// TwinCAT 3 PLC project plc_mrco_vac
// ProgramVersion: 3.1.4022.7
// libraries:
//   LCLS General, * (SLAC)
//   LCLS Vacuum, * (SLAC - LCLS)
//   LCLSVacuumSerialDriverLib, * (SLAC - LCLS)
//   PMPS, * (SLAC - LCLS)
//   Tc2_SerialCom, * (Beckhoff Automation GmbH)
//   Tc2_Standard, * (Beckhoff Automation GmbH)
//   Tc2_System, * (Beckhoff Automation GmbH)
//   Tc3_Module, * (Beckhoff Automation GmbH)
// project tree:
//   / ComTask.TcTTO, PlcTask.TcTTO
//   GVLs/ GVL_COM.TcGVL, GVL_Devices.TcGVL, GVL_PLC_Interfaces.TcGVL, GVL_TC.TcGVL, GVL_Variables.TcGVL
//   POUs/ DIAGNOSTICS.TcPOU, F_Turbo_NC_NO_Valve_Logic.TcPOU, MAIN.TcPOU, PRG_COM.TcPOU, PRG_TC.TcPOU
// real-time tasks:
//   TASK PlcTask: cycle T#10ms, priority 20, ADS port 350
//   TASK ComTask: cycle T#10ms, priority 15, ADS port 351
// I/O:
//   DEVICE Device 1 (EtherCAT), AmsNetId 172.21.132.115.2.1
//     MRCO_PLC_E00_EK1200 [EK1200-5000 EtherCAT Power supply (2A E-Bus)]
//       MRCO_PLC_E01_EL2202
//       MRCO_PLC_E03_EL9184 [EL9184 Potential Connection, 8 x 24V, 8 x Ground]
//       MRCO_PLC_E04_EL6695 [EL6695 EtherCAT Bridge terminal (Primary)]
//       MRCO_PLC_E05_EL9410 [EL9410 E-Bus Power Supplier  (Diagnostics)]
//       MRCO_PLC_E06_EL1004 [EL1004 4Ch. Dig. Input 24V, 3ms]
//       MRCO_PLC_E07_EL2794 [EL2794 4Ch. Dig. Output 24V AC/DC, 2A, short-circuit-proof]
//       MRCO_PLC_E08_EL1004 [EL1004 4Ch. Dig. Input 24V, 3ms]
//       MRCO_PLC_E09_EL2794 [EL2794 4Ch. Dig. Output 24V AC/DC, 2A, short-circuit-proof]
//       MRCO_PLC_E10_EL3318 [EL3318 8Ch. Ana Input Thermocouple (TC)]
//       MRCO_PLC_EXX_EL6070 [EL6070 1Ch. Licensing-Terminal]
//       MRCO_PLC_E11_EL6002 [EL6002 Interface 2Ch. (RS232)]
//       MRCO_PLC_E12_EL6002 [EL6002 Interface 2Ch. (RS232)]
//       MRCO_PLC_E13_EK1122 [EK1122 2 port EtherCAT junction]
//         MRCO_PNL1_EP01_EP2338-0002 [EP2338-0002 8 Ch. Dig. Input/Output 24V, 0,5A, M12]
//         MRCO_PNL1_EP02_EP2624-0002 [EP2624-0002 4Ch. Relay Output, NO (125V AC / 30V DC)]
//         MRCO_PNL1_EP03_EP6002-0002 [EP6002-0002 Interface (RS232/422/485)]
//         MRCO_PNL1_EP04_EP3174-0002 [EP3174-0002 4Ch. Ana. Input +/-10V, 0-10V, 0/4-20mA configurable]
//         MRCO_PNL1_EP05_EP3174-0002 [EP3174-0002 4Ch. Ana. Input +/-10V, 0-10V, 0/4-20mA configurable]
//         MRCO_PNL1_EP06_EP2624-0002
//         MRCO_PNL1_EP07_EP2338-0002 [EP2338-0002 8 Ch. Dig. Input/Output 24V, 0,5A, M12]
//         MRCO_PNL1_EP08_EP2338-0002
//         MRCO_DRL_03 (EK1100) [EK1100 EtherCAT Coupler (2A E-Bus)]
//           MRCO_DRL_03_E01_EL1004
//           MRCO_DRL_03_E02_EL2004 [EL2004 4Ch. Dig. Output 24V, 0.5A]
//           MRCO_DRL_03_E03_EL1004
//           MRCO_DRL_03_E04_EL1004 [EL1004 4Ch. Dig. Input 24V, 3ms]
//           MRCO_DRL_03_E05_EL6001 [EL6001 Interface (RS232)]
//           MRCO_DRL_03_E06_EL2794
//           MRCO_DRL_03_E07_EL1084 [EL1084 4Ch. Dig. Input 24V, 3ms, negative]
//           MRCO_DRL_03_E08_EL9184 [EL9184 Potential Connection, 8 x 24V, 8 x Ground]
//           MRCO_DRL_03_E09_EL9070 [EL9070 Shield terminal]
//           MRCO_DRL_03_E10_EL3174-0002 [EL3174-0002 4Ch. Ana. Input +/-10V, +/-20mA 16 Bit, Isolated Channels]
//           Term 54 (EL9011) [EL9011 End Terminal]
//         VCN_1_VAT590 [590 - All-metal variable leak valve]
// variable links:
//   plc_mrco_vac Instance <-> Device 1 (EtherCAT)/MRCO_PLC_E00_EK1200/MRCO_PLC_E04_EL6695
//     PlcTask Inputs/GVL_PLC_Interfaces.sHUTCH_PLC_NAME <-> IO Inputs/HUTCH_PLC_NAME
//     PlcTask Inputs/GVL_PLC_Interfaces.xEcatBridge_External_device_not_connected <-> SYNC Inputs/External device not connected
//     PlcTask Inputs/GVL_PLC_Interfaces.xEcatBridge_TxPDO_state <-> SYNC Inputs/TxPDO state
//     PlcTask Inputs/GVL_PLC_Interfaces.xEcatBridge_WcState <-> WcState/WcState
//     PlcTask Inputs/GVL_PLC_Interfaces.xTMO_ROUGH1_VRC_01_OPEN_LS <-> IO Inputs/TMO_ROUGH1_VRC_01_OPEN_LS
//     PlcTask Inputs/GVL_PLC_Interfaces.xTMO_ROUGH2_VRC_01_OPEN_LS <-> IO Inputs/TMO_ROUGH2_VRC_01_OPEN_LS
//     PlcTask Outputs/GVL_PLC_Interfaces.rIP1_MAIN_rPRESS <-> IO Outputs/IP1_MAIN_rPRESS
//     PlcTask Outputs/GVL_PLC_Interfaces.sENDSTATION_PLC_NAME <-> IO Outputs/ENDSTATION_PLC_NAME
//     PlcTask Outputs/GVL_PLC_Interfaces.xIP1_HV_SAFETY_ENABLE <-> IO Outputs/IP1_HV_SAFETY_ENABLE
//     PlcTask Outputs/GVL_PLC_Interfaces.xIP1_MAIN_xAT_VAC <-> IO Outputs/IP1_MAIN_xAT_VAC
//     PlcTask Outputs/GVL_PLC_Interfaces.xIP1_MAIN_xPRESS_OK <-> IO Outputs/IP1_MAIN_xPRESS_OK
//     PlcTask Outputs/GVL_PLC_Interfaces.xIP1_ROUGH_VRC_01_OPEN_LS <-> IO Outputs/IP1_ROUGH_VRC_01_OPEN_LS
//     PlcTask Outputs/GVL_PLC_Interfaces.xIP1_ROUGH_VRC_02_OPEN_LS <-> IO Outputs/IP1_ROUGH_VRC_02_OPEN_LS
//     PlcTask Outputs/GVL_PLC_Interfaces.xIP1_ROUGH_VRC_03_OPEN_LS <-> IO Outputs/IP1_ROUGH_VRC_03_OPEN_LS
//     PlcTask Outputs/GVL_PLC_Interfaces.xIP1_TURBOS_ALL_AtSpd <-> IO Outputs/IP1_TURBOS_ALL_AtSpd
//   plc_mrco_vac Instance <-> Device 1 (EtherCAT)/MRCO_PLC_E00_EK1200/MRCO_PLC_E06_EL1004
//     PlcTask Inputs/GVL_Devices.MRCO_MAIN_PTM_01.i_xAtSpd <-> Channel 2/Input
//     PlcTask Inputs/GVL_Devices.MRCO_MAIN_PTM_02.i_xAtSpd <-> Channel 4/Input
//     PlcTask Inputs/GVL_Devices.MRCO_MAIN_PTM_01.i_xFaultNC <-> Channel 1/Input
//     PlcTask Inputs/GVL_Devices.MRCO_MAIN_PTM_02.i_xFaultNC <-> Channel 3/Input
//   plc_mrco_vac Instance <-> Device 1 (EtherCAT)/MRCO_PLC_E00_EK1200/MRCO_PLC_E07_EL2794
//     PlcTask Outputs/GVL_Devices.MRCO_MAIN_PTM_01.q_RunDO <-> Channel 1/Output
//     PlcTask Outputs/GVL_Devices.MRCO_MAIN_PTM_02.q_RunDO <-> Channel 3/Output
//     PlcTask Outputs/GVL_Devices.MRCO_MAIN_PTM_03.q_RunDO <-> Channel 2/Output
//     PlcTask Outputs/GVL_Devices.MRCO_MAIN_PTM_04.q_RunDO <-> Channel 4/Output
//   plc_mrco_vac Instance <-> Device 1 (EtherCAT)/MRCO_PLC_E00_EK1200/MRCO_PLC_E08_EL1004
//     PlcTask Inputs/GVL_Devices.MRCO_MAIN_PTM_03.i_xAtSpd <-> Channel 2/Input
//     PlcTask Inputs/GVL_Devices.MRCO_MAIN_PTM_04.i_xAtSpd <-> Channel 4/Input
//     PlcTask Inputs/GVL_Devices.MRCO_MAIN_PTM_03.i_xFaultNC <-> Channel 1/Input
//     PlcTask Inputs/GVL_Devices.MRCO_MAIN_PTM_04.i_xFaultNC <-> Channel 3/Input
//   plc_mrco_vac Instance <-> Device 1 (EtherCAT)/MRCO_PLC_E00_EK1200/MRCO_PLC_E09_EL2794
//     PlcTask Outputs/GVL_PLC_Interfaces.xHighVoltageSafteyLoopEnable <-> Channel 1/Output
//   plc_mrco_vac Instance <-> Device 1 (EtherCAT)/MRCO_PLC_E00_EK1200/MRCO_PLC_E10_EL3318
//     PlcTask Inputs/GVL_TC.TC_01.bError <-> TC Channel 1/Status/Error
//     PlcTask Inputs/GVL_TC.TC_02.bError <-> TC Channel 2/Status/Error
//     PlcTask Inputs/GVL_TC.TC_03.bError <-> TC Channel 3/Status/Error
//     PlcTask Inputs/GVL_TC.TC_04.bError <-> TC Channel 4/Status/Error
//     PlcTask Inputs/GVL_TC.TC_05.bError <-> TC Channel 5/Status/Error
//     PlcTask Inputs/GVL_TC.TC_06.bError <-> TC Channel 6/Status/Error
//     PlcTask Inputs/GVL_TC.TC_07.bError <-> TC Channel 7/Status/Error
//     PlcTask Inputs/GVL_TC.TC_08.bError <-> TC Channel 8/Status/Error
//     PlcTask Inputs/GVL_TC.TC_01.bOverrange <-> TC Channel 1/Status/Overrange
//     PlcTask Inputs/GVL_TC.TC_02.bOverrange <-> TC Channel 2/Status/Overrange
//     PlcTask Inputs/GVL_TC.TC_03.bOverrange <-> TC Channel 3/Status/Overrange
//     PlcTask Inputs/GVL_TC.TC_04.bOverrange <-> TC Channel 4/Status/Overrange
//     PlcTask Inputs/GVL_TC.TC_05.bOverrange <-> TC Channel 5/Status/Overrange
//     PlcTask Inputs/GVL_TC.TC_06.bOverrange <-> TC Channel 6/Status/Overrange
//     PlcTask Inputs/GVL_TC.TC_07.bOverrange <-> TC Channel 7/Status/Overrange
//     PlcTask Inputs/GVL_TC.TC_08.bOverrange <-> TC Channel 8/Status/Overrange
//     PlcTask Inputs/GVL_TC.TC_01.bUnderrange <-> TC Channel 1/Status/Underrange
//     PlcTask Inputs/GVL_TC.TC_02.bUnderrange <-> TC Channel 2/Status/Underrange
//     PlcTask Inputs/GVL_TC.TC_03.bUnderrange <-> TC Channel 3/Status/Underrange
//     PlcTask Inputs/GVL_TC.TC_04.bUnderrange <-> TC Channel 4/Status/Underrange
//     PlcTask Inputs/GVL_TC.TC_05.bUnderrange <-> TC Channel 5/Status/Underrange
//     PlcTask Inputs/GVL_TC.TC_06.bUnderrange <-> TC Channel 6/Status/Underrange
//     PlcTask Inputs/GVL_TC.TC_07.bUnderrange <-> TC Channel 7/Status/Underrange
//     PlcTask Inputs/GVL_TC.TC_08.bUnderrange <-> TC Channel 8/Status/Underrange
//     PlcTask Inputs/GVL_TC.TC_01.iRaw <-> TC Channel 1/Value
//     PlcTask Inputs/GVL_TC.TC_02.iRaw <-> TC Channel 2/Value
//     PlcTask Inputs/GVL_TC.TC_03.iRaw <-> TC Channel 3/Value
//     PlcTask Inputs/GVL_TC.TC_04.iRaw <-> TC Channel 4/Value
//     PlcTask Inputs/GVL_TC.TC_05.iRaw <-> TC Channel 5/Value
//     PlcTask Inputs/GVL_TC.TC_06.iRaw <-> TC Channel 6/Value
//     PlcTask Inputs/GVL_TC.TC_07.iRaw <-> TC Channel 7/Value
//     PlcTask Inputs/GVL_TC.TC_08.iRaw <-> TC Channel 8/Value
//   plc_mrco_vac Instance <-> Device 1 (EtherCAT)/MRCO_PLC_E00_EK1200/MRCO_PLC_E11_EL6002
//     ComTask Inputs/GVL_COM.stComIn_MRCO_MAIN_PTM_01/D[0] <-> COM TxPDO-Map Inputs Channel 1/Data In 0
//     ComTask Inputs/GVL_COM.stComIn_MRCO_MAIN_PTM_01/D[10] <-> COM TxPDO-Map Inputs Channel 1/Data In 10
//     ComTask Inputs/GVL_COM.stComIn_MRCO_MAIN_PTM_01/D[11] <-> COM TxPDO-Map Inputs Channel 1/Data In 11
//     ComTask Inputs/GVL_COM.stComIn_MRCO_MAIN_PTM_01/D[12] <-> COM TxPDO-Map Inputs Channel 1/Data In 12
//     ComTask Inputs/GVL_COM.stComIn_MRCO_MAIN_PTM_01/D[13] <-> COM TxPDO-Map Inputs Channel 1/Data In 13
//     ComTask Inputs/GVL_COM.stComIn_MRCO_MAIN_PTM_01/D[14] <-> COM TxPDO-Map Inputs Channel 1/Data In 14
//     ComTask Inputs/GVL_COM.stComIn_MRCO_MAIN_PTM_01/D[15] <-> COM TxPDO-Map Inputs Channel 1/Data In 15
//     ComTask Inputs/GVL_COM.stComIn_MRCO_MAIN_PTM_01/D[16] <-> COM TxPDO-Map Inputs Channel 1/Data In 16
//     ComTask Inputs/GVL_COM.stComIn_MRCO_MAIN_PTM_01/D[17] <-> COM TxPDO-Map Inputs Channel 1/Data In 17
//     ComTask Inputs/GVL_COM.stComIn_MRCO_MAIN_PTM_01/D[18] <-> COM TxPDO-Map Inputs Channel 1/Data In 18
//     ComTask Inputs/GVL_COM.stComIn_MRCO_MAIN_PTM_01/D[19] <-> COM TxPDO-Map Inputs Channel 1/Data In 19
//     ComTask Inputs/GVL_COM.stComIn_MRCO_MAIN_PTM_01/D[1] <-> COM TxPDO-Map Inputs Channel 1/Data In 1
//     ComTask Inputs/GVL_COM.stComIn_MRCO_MAIN_PTM_01/D[20] <-> COM TxPDO-Map Inputs Channel 1/Data In 20
//     ComTask Inputs/GVL_COM.stComIn_MRCO_MAIN_PTM_01/D[21] <-> COM TxPDO-Map Inputs Channel 1/Data In 21
//     ComTask Inputs/GVL_COM.stComIn_MRCO_MAIN_PTM_01/D[2] <-> COM TxPDO-Map Inputs Channel 1/Data In 2
//     ComTask Inputs/GVL_COM.stComIn_MRCO_MAIN_PTM_01/D[3] <-> COM TxPDO-Map Inputs Channel 1/Data In 3
//     ComTask Inputs/GVL_COM.stComIn_MRCO_MAIN_PTM_01/D[4] <-> COM TxPDO-Map Inputs Channel 1/Data In 4
//     ComTask Inputs/GVL_COM.stComIn_MRCO_MAIN_PTM_01/D[5] <-> COM TxPDO-Map Inputs Channel 1/Data In 5
//     ComTask Inputs/GVL_COM.stComIn_MRCO_MAIN_PTM_01/D[6] <-> COM TxPDO-Map Inputs Channel 1/Data In 6
//     ComTask Inputs/GVL_COM.stComIn_MRCO_MAIN_PTM_01/D[7] <-> COM TxPDO-Map Inputs Channel 1/Data In 7
//     ComTask Inputs/GVL_COM.stComIn_MRCO_MAIN_PTM_01/D[8] <-> COM TxPDO-Map Inputs Channel 1/Data In 8
//     ComTask Inputs/GVL_COM.stComIn_MRCO_MAIN_PTM_01/D[9] <-> COM TxPDO-Map Inputs Channel 1/Data In 9
//     ComTask Inputs/GVL_COM.stComIn_MRCO_MAIN_PTM_03/D[0] <-> COM TxPDO-Map Inputs Channel 2/Data In 0
//     ComTask Inputs/GVL_COM.stComIn_MRCO_MAIN_PTM_03/D[10] <-> COM TxPDO-Map Inputs Channel 2/Data In 10
//     ComTask Inputs/GVL_COM.stComIn_MRCO_MAIN_PTM_03/D[11] <-> COM TxPDO-Map Inputs Channel 2/Data In 11
//     ComTask Inputs/GVL_COM.stComIn_MRCO_MAIN_PTM_03/D[12] <-> COM TxPDO-Map Inputs Channel 2/Data In 12
//     ComTask Inputs/GVL_COM.stComIn_MRCO_MAIN_PTM_03/D[13] <-> COM TxPDO-Map Inputs Channel 2/Data In 13
//     ComTask Inputs/GVL_COM.stComIn_MRCO_MAIN_PTM_03/D[14] <-> COM TxPDO-Map Inputs Channel 2/Data In 14
//     ComTask Inputs/GVL_COM.stComIn_MRCO_MAIN_PTM_03/D[15] <-> COM TxPDO-Map Inputs Channel 2/Data In 15
//     ComTask Inputs/GVL_COM.stComIn_MRCO_MAIN_PTM_03/D[16] <-> COM TxPDO-Map Inputs Channel 2/Data In 16
//     ComTask Inputs/GVL_COM.stComIn_MRCO_MAIN_PTM_03/D[17] <-> COM TxPDO-Map Inputs Channel 2/Data In 17
//     ComTask Inputs/GVL_COM.stComIn_MRCO_MAIN_PTM_03/D[18] <-> COM TxPDO-Map Inputs Channel 2/Data In 18
//     ComTask Inputs/GVL_COM.stComIn_MRCO_MAIN_PTM_03/D[19] <-> COM TxPDO-Map Inputs Channel 2/Data In 19
//     ComTask Inputs/GVL_COM.stComIn_MRCO_MAIN_PTM_03/D[1] <-> COM TxPDO-Map Inputs Channel 2/Data In 1
//     ComTask Inputs/GVL_COM.stComIn_MRCO_MAIN_PTM_03/D[20] <-> COM TxPDO-Map Inputs Channel 2/Data In 20
//     ComTask Inputs/GVL_COM.stComIn_MRCO_MAIN_PTM_03/D[21] <-> COM TxPDO-Map Inputs Channel 2/Data In 21
//     ComTask Inputs/GVL_COM.stComIn_MRCO_MAIN_PTM_03/D[2] <-> COM TxPDO-Map Inputs Channel 2/Data In 2
//     ComTask Inputs/GVL_COM.stComIn_MRCO_MAIN_PTM_03/D[3] <-> COM TxPDO-Map Inputs Channel 2/Data In 3
//     ComTask Inputs/GVL_COM.stComIn_MRCO_MAIN_PTM_03/D[4] <-> COM TxPDO-Map Inputs Channel 2/Data In 4
//     ComTask Inputs/GVL_COM.stComIn_MRCO_MAIN_PTM_03/D[5] <-> COM TxPDO-Map Inputs Channel 2/Data In 5
//     ComTask Inputs/GVL_COM.stComIn_MRCO_MAIN_PTM_03/D[6] <-> COM TxPDO-Map Inputs Channel 2/Data In 6
//     ComTask Inputs/GVL_COM.stComIn_MRCO_MAIN_PTM_03/D[7] <-> COM TxPDO-Map Inputs Channel 2/Data In 7
//     ComTask Inputs/GVL_COM.stComIn_MRCO_MAIN_PTM_03/D[8] <-> COM TxPDO-Map Inputs Channel 2/Data In 8
//     ComTask Inputs/GVL_COM.stComIn_MRCO_MAIN_PTM_03/D[9] <-> COM TxPDO-Map Inputs Channel 2/Data In 9
//     ComTask Inputs/GVL_COM.stComIn_MRCO_MAIN_PTM_01/Status <-> COM TxPDO-Map Inputs Channel 1/Status
//     ComTask Inputs/GVL_COM.stComIn_MRCO_MAIN_PTM_03/Status <-> COM TxPDO-Map Inputs Channel 2/Status
//     ComTask Outputs/GVL_COM.stComOut_MRCO_MAIN_PTM_01/Ctrl <-> COM RxPDO-Map Outputs Channel 1/Ctrl
//     ComTask Outputs/GVL_COM.stComOut_MRCO_MAIN_PTM_03/Ctrl <-> COM RxPDO-Map Outputs Channel 2/Ctrl
//     ComTask Outputs/GVL_COM.stComOut_MRCO_MAIN_PTM_01/D[0] <-> COM RxPDO-Map Outputs Channel 1/Data Out 0
//     ComTask Outputs/GVL_COM.stComOut_MRCO_MAIN_PTM_01/D[10] <-> COM RxPDO-Map Outputs Channel 1/Data Out 10
//     ComTask Outputs/GVL_COM.stComOut_MRCO_MAIN_PTM_01/D[11] <-> COM RxPDO-Map Outputs Channel 1/Data Out 11
//     ComTask Outputs/GVL_COM.stComOut_MRCO_MAIN_PTM_01/D[12] <-> COM RxPDO-Map Outputs Channel 1/Data Out 12
//     ComTask Outputs/GVL_COM.stComOut_MRCO_MAIN_PTM_01/D[13] <-> COM RxPDO-Map Outputs Channel 1/Data Out 13
//     ComTask Outputs/GVL_COM.stComOut_MRCO_MAIN_PTM_01/D[14] <-> COM RxPDO-Map Outputs Channel 1/Data Out 14
//     ComTask Outputs/GVL_COM.stComOut_MRCO_MAIN_PTM_01/D[15] <-> COM RxPDO-Map Outputs Channel 1/Data Out 15
//     ComTask Outputs/GVL_COM.stComOut_MRCO_MAIN_PTM_01/D[16] <-> COM RxPDO-Map Outputs Channel 1/Data Out 16
//     ComTask Outputs/GVL_COM.stComOut_MRCO_MAIN_PTM_01/D[17] <-> COM RxPDO-Map Outputs Channel 1/Data Out 17
//     ComTask Outputs/GVL_COM.stComOut_MRCO_MAIN_PTM_01/D[18] <-> COM RxPDO-Map Outputs Channel 1/Data Out 18
//     ComTask Outputs/GVL_COM.stComOut_MRCO_MAIN_PTM_01/D[19] <-> COM RxPDO-Map Outputs Channel 1/Data Out 19
//     ComTask Outputs/GVL_COM.stComOut_MRCO_MAIN_PTM_01/D[1] <-> COM RxPDO-Map Outputs Channel 1/Data Out 1
//     ComTask Outputs/GVL_COM.stComOut_MRCO_MAIN_PTM_01/D[20] <-> COM RxPDO-Map Outputs Channel 1/Data Out 20
//     ComTask Outputs/GVL_COM.stComOut_MRCO_MAIN_PTM_01/D[21] <-> COM RxPDO-Map Outputs Channel 1/Data Out 21
//     ComTask Outputs/GVL_COM.stComOut_MRCO_MAIN_PTM_01/D[2] <-> COM RxPDO-Map Outputs Channel 1/Data Out 2
//     ComTask Outputs/GVL_COM.stComOut_MRCO_MAIN_PTM_01/D[3] <-> COM RxPDO-Map Outputs Channel 1/Data Out 3
//     ComTask Outputs/GVL_COM.stComOut_MRCO_MAIN_PTM_01/D[4] <-> COM RxPDO-Map Outputs Channel 1/Data Out 4
//     ComTask Outputs/GVL_COM.stComOut_MRCO_MAIN_PTM_01/D[5] <-> COM RxPDO-Map Outputs Channel 1/Data Out 5
//     ComTask Outputs/GVL_COM.stComOut_MRCO_MAIN_PTM_01/D[6] <-> COM RxPDO-Map Outputs Channel 1/Data Out 6
//     ComTask Outputs/GVL_COM.stComOut_MRCO_MAIN_PTM_01/D[7] <-> COM RxPDO-Map Outputs Channel 1/Data Out 7
//     ComTask Outputs/GVL_COM.stComOut_MRCO_MAIN_PTM_01/D[8] <-> COM RxPDO-Map Outputs Channel 1/Data Out 8
//     ComTask Outputs/GVL_COM.stComOut_MRCO_MAIN_PTM_01/D[9] <-> COM RxPDO-Map Outputs Channel 1/Data Out 9
//     ComTask Outputs/GVL_COM.stComOut_MRCO_MAIN_PTM_03/D[0] <-> COM RxPDO-Map Outputs Channel 2/Data Out 0
//     ComTask Outputs/GVL_COM.stComOut_MRCO_MAIN_PTM_03/D[10] <-> COM RxPDO-Map Outputs Channel 2/Data Out 10
//     ComTask Outputs/GVL_COM.stComOut_MRCO_MAIN_PTM_03/D[11] <-> COM RxPDO-Map Outputs Channel 2/Data Out 11
//     ComTask Outputs/GVL_COM.stComOut_MRCO_MAIN_PTM_03/D[12] <-> COM RxPDO-Map Outputs Channel 2/Data Out 12
//     ComTask Outputs/GVL_COM.stComOut_MRCO_MAIN_PTM_03/D[13] <-> COM RxPDO-Map Outputs Channel 2/Data Out 13
//     ComTask Outputs/GVL_COM.stComOut_MRCO_MAIN_PTM_03/D[14] <-> COM RxPDO-Map Outputs Channel 2/Data Out 14
//     ComTask Outputs/GVL_COM.stComOut_MRCO_MAIN_PTM_03/D[15] <-> COM RxPDO-Map Outputs Channel 2/Data Out 15
//     ComTask Outputs/GVL_COM.stComOut_MRCO_MAIN_PTM_03/D[16] <-> COM RxPDO-Map Outputs Channel 2/Data Out 16
//     ComTask Outputs/GVL_COM.stComOut_MRCO_MAIN_PTM_03/D[17] <-> COM RxPDO-Map Outputs Channel 2/Data Out 17
//     ComTask Outputs/GVL_COM.stComOut_MRCO_MAIN_PTM_03/D[18] <-> COM RxPDO-Map Outputs Channel 2/Data Out 18
//     ComTask Outputs/GVL_COM.stComOut_MRCO_MAIN_PTM_03/D[19] <-> COM RxPDO-Map Outputs Channel 2/Data Out 19
//     ComTask Outputs/GVL_COM.stComOut_MRCO_MAIN_PTM_03/D[1] <-> COM RxPDO-Map Outputs Channel 2/Data Out 1
//     ComTask Outputs/GVL_COM.stComOut_MRCO_MAIN_PTM_03/D[20] <-> COM RxPDO-Map Outputs Channel 2/Data Out 20
//     ComTask Outputs/GVL_COM.stComOut_MRCO_MAIN_PTM_03/D[21] <-> COM RxPDO-Map Outputs Channel 2/Data Out 21
//     ComTask Outputs/GVL_COM.stComOut_MRCO_MAIN_PTM_03/D[2] <-> COM RxPDO-Map Outputs Channel 2/Data Out 2
//     ComTask Outputs/GVL_COM.stComOut_MRCO_MAIN_PTM_03/D[3] <-> COM RxPDO-Map Outputs Channel 2/Data Out 3
//     ComTask Outputs/GVL_COM.stComOut_MRCO_MAIN_PTM_03/D[4] <-> COM RxPDO-Map Outputs Channel 2/Data Out 4
//     ComTask Outputs/GVL_COM.stComOut_MRCO_MAIN_PTM_03/D[5] <-> COM RxPDO-Map Outputs Channel 2/Data Out 5
//     ComTask Outputs/GVL_COM.stComOut_MRCO_MAIN_PTM_03/D[6] <-> COM RxPDO-Map Outputs Channel 2/Data Out 6
//     ComTask Outputs/GVL_COM.stComOut_MRCO_MAIN_PTM_03/D[7] <-> COM RxPDO-Map Outputs Channel 2/Data Out 7
//     ComTask Outputs/GVL_COM.stComOut_MRCO_MAIN_PTM_03/D[8] <-> COM RxPDO-Map Outputs Channel 2/Data Out 8
//     ComTask Outputs/GVL_COM.stComOut_MRCO_MAIN_PTM_03/D[9] <-> COM RxPDO-Map Outputs Channel 2/Data Out 9
//   plc_mrco_vac Instance <-> Device 1 (EtherCAT)/MRCO_PLC_E00_EK1200/MRCO_PLC_E12_EL6002
//     ComTask Inputs/GVL_COM.stComIn_MRCO_MAIN_PTM_02/D[0] <-> COM TxPDO-Map Inputs Channel 1/Data In 0
//     ComTask Inputs/GVL_COM.stComIn_MRCO_MAIN_PTM_02/D[10] <-> COM TxPDO-Map Inputs Channel 1/Data In 10
//     ComTask Inputs/GVL_COM.stComIn_MRCO_MAIN_PTM_02/D[11] <-> COM TxPDO-Map Inputs Channel 1/Data In 11
//     ComTask Inputs/GVL_COM.stComIn_MRCO_MAIN_PTM_02/D[12] <-> COM TxPDO-Map Inputs Channel 1/Data In 12
//     ComTask Inputs/GVL_COM.stComIn_MRCO_MAIN_PTM_02/D[13] <-> COM TxPDO-Map Inputs Channel 1/Data In 13
//     ComTask Inputs/GVL_COM.stComIn_MRCO_MAIN_PTM_02/D[14] <-> COM TxPDO-Map Inputs Channel 1/Data In 14
//     ComTask Inputs/GVL_COM.stComIn_MRCO_MAIN_PTM_02/D[15] <-> COM TxPDO-Map Inputs Channel 1/Data In 15
//     ComTask Inputs/GVL_COM.stComIn_MRCO_MAIN_PTM_02/D[16] <-> COM TxPDO-Map Inputs Channel 1/Data In 16
//     ComTask Inputs/GVL_COM.stComIn_MRCO_MAIN_PTM_02/D[17] <-> COM TxPDO-Map Inputs Channel 1/Data In 17
//     ComTask Inputs/GVL_COM.stComIn_MRCO_MAIN_PTM_02/D[18] <-> COM TxPDO-Map Inputs Channel 1/Data In 18
//     ComTask Inputs/GVL_COM.stComIn_MRCO_MAIN_PTM_02/D[19] <-> COM TxPDO-Map Inputs Channel 1/Data In 19
//     ComTask Inputs/GVL_COM.stComIn_MRCO_MAIN_PTM_02/D[1] <-> COM TxPDO-Map Inputs Channel 1/Data In 1
//     ComTask Inputs/GVL_COM.stComIn_MRCO_MAIN_PTM_02/D[20] <-> COM TxPDO-Map Inputs Channel 1/Data In 20
//     ComTask Inputs/GVL_COM.stComIn_MRCO_MAIN_PTM_02/D[21] <-> COM TxPDO-Map Inputs Channel 1/Data In 21
//     ComTask Inputs/GVL_COM.stComIn_MRCO_MAIN_PTM_02/D[2] <-> COM TxPDO-Map Inputs Channel 1/Data In 2
//     ComTask Inputs/GVL_COM.stComIn_MRCO_MAIN_PTM_02/D[3] <-> COM TxPDO-Map Inputs Channel 1/Data In 3
//     ComTask Inputs/GVL_COM.stComIn_MRCO_MAIN_PTM_02/D[4] <-> COM TxPDO-Map Inputs Channel 1/Data In 4
//     ComTask Inputs/GVL_COM.stComIn_MRCO_MAIN_PTM_02/D[5] <-> COM TxPDO-Map Inputs Channel 1/Data In 5
//     ComTask Inputs/GVL_COM.stComIn_MRCO_MAIN_PTM_02/D[6] <-> COM TxPDO-Map Inputs Channel 1/Data In 6
//     ComTask Inputs/GVL_COM.stComIn_MRCO_MAIN_PTM_02/D[7] <-> COM TxPDO-Map Inputs Channel 1/Data In 7
//     ComTask Inputs/GVL_COM.stComIn_MRCO_MAIN_PTM_02/D[8] <-> COM TxPDO-Map Inputs Channel 1/Data In 8
//     ComTask Inputs/GVL_COM.stComIn_MRCO_MAIN_PTM_02/D[9] <-> COM TxPDO-Map Inputs Channel 1/Data In 9
//     ComTask Inputs/GVL_COM.stComIn_MRCO_MAIN_PTM_04/D[0] <-> COM TxPDO-Map Inputs Channel 2/Data In 0
//     ComTask Inputs/GVL_COM.stComIn_MRCO_MAIN_PTM_04/D[10] <-> COM TxPDO-Map Inputs Channel 2/Data In 10
//     ComTask Inputs/GVL_COM.stComIn_MRCO_MAIN_PTM_04/D[11] <-> COM TxPDO-Map Inputs Channel 2/Data In 11
//     ComTask Inputs/GVL_COM.stComIn_MRCO_MAIN_PTM_04/D[12] <-> COM TxPDO-Map Inputs Channel 2/Data In 12
//     ComTask Inputs/GVL_COM.stComIn_MRCO_MAIN_PTM_04/D[13] <-> COM TxPDO-Map Inputs Channel 2/Data In 13
//     ComTask Inputs/GVL_COM.stComIn_MRCO_MAIN_PTM_04/D[14] <-> COM TxPDO-Map Inputs Channel 2/Data In 14
//     ComTask Inputs/GVL_COM.stComIn_MRCO_MAIN_PTM_04/D[15] <-> COM TxPDO-Map Inputs Channel 2/Data In 15
//     ComTask Inputs/GVL_COM.stComIn_MRCO_MAIN_PTM_04/D[16] <-> COM TxPDO-Map Inputs Channel 2/Data In 16
//     ComTask Inputs/GVL_COM.stComIn_MRCO_MAIN_PTM_04/D[17] <-> COM TxPDO-Map Inputs Channel 2/Data In 17
//     ComTask Inputs/GVL_COM.stComIn_MRCO_MAIN_PTM_04/D[18] <-> COM TxPDO-Map Inputs Channel 2/Data In 18
//     ComTask Inputs/GVL_COM.stComIn_MRCO_MAIN_PTM_04/D[19] <-> COM TxPDO-Map Inputs Channel 2/Data In 19
//     ComTask Inputs/GVL_COM.stComIn_MRCO_MAIN_PTM_04/D[1] <-> COM TxPDO-Map Inputs Channel 2/Data In 1
//     ComTask Inputs/GVL_COM.stComIn_MRCO_MAIN_PTM_04/D[20] <-> COM TxPDO-Map Inputs Channel 2/Data In 20
//     ComTask Inputs/GVL_COM.stComIn_MRCO_MAIN_PTM_04/D[21] <-> COM TxPDO-Map Inputs Channel 2/Data In 21
//     ComTask Inputs/GVL_COM.stComIn_MRCO_MAIN_PTM_04/D[2] <-> COM TxPDO-Map Inputs Channel 2/Data In 2
//     ComTask Inputs/GVL_COM.stComIn_MRCO_MAIN_PTM_04/D[3] <-> COM TxPDO-Map Inputs Channel 2/Data In 3
//     ComTask Inputs/GVL_COM.stComIn_MRCO_MAIN_PTM_04/D[4] <-> COM TxPDO-Map Inputs Channel 2/Data In 4
//     ComTask Inputs/GVL_COM.stComIn_MRCO_MAIN_PTM_04/D[5] <-> COM TxPDO-Map Inputs Channel 2/Data In 5
//     ComTask Inputs/GVL_COM.stComIn_MRCO_MAIN_PTM_04/D[6] <-> COM TxPDO-Map Inputs Channel 2/Data In 6
//     ComTask Inputs/GVL_COM.stComIn_MRCO_MAIN_PTM_04/D[7] <-> COM TxPDO-Map Inputs Channel 2/Data In 7
//     ComTask Inputs/GVL_COM.stComIn_MRCO_MAIN_PTM_04/D[8] <-> COM TxPDO-Map Inputs Channel 2/Data In 8
//     ComTask Inputs/GVL_COM.stComIn_MRCO_MAIN_PTM_04/D[9] <-> COM TxPDO-Map Inputs Channel 2/Data In 9
//     ComTask Inputs/GVL_COM.stComIn_MRCO_MAIN_PTM_02/Status <-> COM TxPDO-Map Inputs Channel 1/Status
//     ComTask Inputs/GVL_COM.stComIn_MRCO_MAIN_PTM_04/Status <-> COM TxPDO-Map Inputs Channel 2/Status
//     ComTask Outputs/GVL_COM.stComOut_MRCO_MAIN_PTM_02/Ctrl <-> COM RxPDO-Map Outputs Channel 1/Ctrl
//     ComTask Outputs/GVL_COM.stComOut_MRCO_MAIN_PTM_04/Ctrl <-> COM RxPDO-Map Outputs Channel 2/Ctrl
//     ComTask Outputs/GVL_COM.stComOut_MRCO_MAIN_PTM_02/D[10] <-> COM RxPDO-Map Outputs Channel 1/Data Out 10
//     ComTask Outputs/GVL_COM.stComOut_MRCO_MAIN_PTM_02/D[11] <-> COM RxPDO-Map Outputs Channel 1/Data Out 11
//     ComTask Outputs/GVL_COM.stComOut_MRCO_MAIN_PTM_02/D[12] <-> COM RxPDO-Map Outputs Channel 1/Data Out 12
//     ComTask Outputs/GVL_COM.stComOut_MRCO_MAIN_PTM_02/D[13] <-> COM RxPDO-Map Outputs Channel 1/Data Out 13
//     ComTask Outputs/GVL_COM.stComOut_MRCO_MAIN_PTM_02/D[14] <-> COM RxPDO-Map Outputs Channel 1/Data Out 14
//     ComTask Outputs/GVL_COM.stComOut_MRCO_MAIN_PTM_02/D[15] <-> COM RxPDO-Map Outputs Channel 1/Data Out 15
//     ComTask Outputs/GVL_COM.stComOut_MRCO_MAIN_PTM_02/D[16] <-> COM RxPDO-Map Outputs Channel 1/Data Out 16
//     ComTask Outputs/GVL_COM.stComOut_MRCO_MAIN_PTM_02/D[17] <-> COM RxPDO-Map Outputs Channel 1/Data Out 17
//     ComTask Outputs/GVL_COM.stComOut_MRCO_MAIN_PTM_02/D[18] <-> COM RxPDO-Map Outputs Channel 1/Data Out 18
//     ComTask Outputs/GVL_COM.stComOut_MRCO_MAIN_PTM_02/D[19] <-> COM RxPDO-Map Outputs Channel 1/Data Out 19
//     ComTask Outputs/GVL_COM.stComOut_MRCO_MAIN_PTM_02/D[1] <-> COM RxPDO-Map Outputs Channel 1/Data Out 1
//     ComTask Outputs/GVL_COM.stComOut_MRCO_MAIN_PTM_02/D[20] <-> COM RxPDO-Map Outputs Channel 1/Data Out 20
//     ComTask Outputs/GVL_COM.stComOut_MRCO_MAIN_PTM_02/D[21] <-> COM RxPDO-Map Outputs Channel 1/Data Out 21
//     ComTask Outputs/GVL_COM.stComOut_MRCO_MAIN_PTM_02/D[2] <-> COM RxPDO-Map Outputs Channel 1/Data Out 2
//     ComTask Outputs/GVL_COM.stComOut_MRCO_MAIN_PTM_02/D[3] <-> COM RxPDO-Map Outputs Channel 1/Data Out 3
//     ComTask Outputs/GVL_COM.stComOut_MRCO_MAIN_PTM_02/D[4] <-> COM RxPDO-Map Outputs Channel 1/Data Out 4
//     ComTask Outputs/GVL_COM.stComOut_MRCO_MAIN_PTM_02/D[5] <-> COM RxPDO-Map Outputs Channel 1/Data Out 5
//     ComTask Outputs/GVL_COM.stComOut_MRCO_MAIN_PTM_02/D[6] <-> COM RxPDO-Map Outputs Channel 1/Data Out 6
//     ComTask Outputs/GVL_COM.stComOut_MRCO_MAIN_PTM_02/D[7] <-> COM RxPDO-Map Outputs Channel 1/Data Out 7
//     ComTask Outputs/GVL_COM.stComOut_MRCO_MAIN_PTM_02/D[8] <-> COM RxPDO-Map Outputs Channel 1/Data Out 8
//     ComTask Outputs/GVL_COM.stComOut_MRCO_MAIN_PTM_02/D[9] <-> COM RxPDO-Map Outputs Channel 1/Data Out 9
//     ComTask Outputs/GVL_COM.stComOut_MRCO_MAIN_PTM_04/D[0] <-> COM RxPDO-Map Outputs Channel 2/Data Out 0
//     ComTask Outputs/GVL_COM.stComOut_MRCO_MAIN_PTM_04/D[10] <-> COM RxPDO-Map Outputs Channel 2/Data Out 10
//     ComTask Outputs/GVL_COM.stComOut_MRCO_MAIN_PTM_04/D[11] <-> COM RxPDO-Map Outputs Channel 2/Data Out 11
//     ComTask Outputs/GVL_COM.stComOut_MRCO_MAIN_PTM_04/D[12] <-> COM RxPDO-Map Outputs Channel 2/Data Out 12
//     ComTask Outputs/GVL_COM.stComOut_MRCO_MAIN_PTM_04/D[13] <-> COM RxPDO-Map Outputs Channel 2/Data Out 13
//     ComTask Outputs/GVL_COM.stComOut_MRCO_MAIN_PTM_04/D[14] <-> COM RxPDO-Map Outputs Channel 2/Data Out 14
//     ComTask Outputs/GVL_COM.stComOut_MRCO_MAIN_PTM_04/D[15] <-> COM RxPDO-Map Outputs Channel 2/Data Out 15
//     ComTask Outputs/GVL_COM.stComOut_MRCO_MAIN_PTM_04/D[16] <-> COM RxPDO-Map Outputs Channel 2/Data Out 16
//     ComTask Outputs/GVL_COM.stComOut_MRCO_MAIN_PTM_04/D[17] <-> COM RxPDO-Map Outputs Channel 2/Data Out 17
//     ComTask Outputs/GVL_COM.stComOut_MRCO_MAIN_PTM_04/D[18] <-> COM RxPDO-Map Outputs Channel 2/Data Out 18
//     ComTask Outputs/GVL_COM.stComOut_MRCO_MAIN_PTM_04/D[19] <-> COM RxPDO-Map Outputs Channel 2/Data Out 19
//     ComTask Outputs/GVL_COM.stComOut_MRCO_MAIN_PTM_04/D[1] <-> COM RxPDO-Map Outputs Channel 2/Data Out 1
//     ComTask Outputs/GVL_COM.stComOut_MRCO_MAIN_PTM_04/D[20] <-> COM RxPDO-Map Outputs Channel 2/Data Out 20
//     ComTask Outputs/GVL_COM.stComOut_MRCO_MAIN_PTM_04/D[21] <-> COM RxPDO-Map Outputs Channel 2/Data Out 21
//     ComTask Outputs/GVL_COM.stComOut_MRCO_MAIN_PTM_04/D[2] <-> COM RxPDO-Map Outputs Channel 2/Data Out 2
//     ComTask Outputs/GVL_COM.stComOut_MRCO_MAIN_PTM_04/D[3] <-> COM RxPDO-Map Outputs Channel 2/Data Out 3
//     ComTask Outputs/GVL_COM.stComOut_MRCO_MAIN_PTM_04/D[4] <-> COM RxPDO-Map Outputs Channel 2/Data Out 4
//     ComTask Outputs/GVL_COM.stComOut_MRCO_MAIN_PTM_04/D[5] <-> COM RxPDO-Map Outputs Channel 2/Data Out 5
//     ComTask Outputs/GVL_COM.stComOut_MRCO_MAIN_PTM_04/D[6] <-> COM RxPDO-Map Outputs Channel 2/Data Out 6
//     ComTask Outputs/GVL_COM.stComOut_MRCO_MAIN_PTM_04/D[7] <-> COM RxPDO-Map Outputs Channel 2/Data Out 7
//     ComTask Outputs/GVL_COM.stComOut_MRCO_MAIN_PTM_04/D[8] <-> COM RxPDO-Map Outputs Channel 2/Data Out 8
//     ComTask Outputs/GVL_COM.stComOut_MRCO_MAIN_PTM_04/D[9] <-> COM RxPDO-Map Outputs Channel 2/Data Out 9
//   plc_mrco_vac Instance <-> Device 1 (EtherCAT)/MRCO_PLC_E00_EK1200/MRCO_PLC_E13_EK1122/MRCO_DRL_03 (EK1100)/MRCO_DRL_03_E01_EL1004
//     PlcTask Inputs/GVL_Devices.MRCO_MSC_VRC_01.i_xClsLS <-> Channel 2/Input
//     PlcTask Inputs/GVL_Devices.MRCO_MSC_VRC_01.i_xOpnLS <-> Channel 1/Input
//     PlcTask Inputs/GVL_Devices.MRCO_ROUGH_VRC_04.i_xClsLS <-> Channel 4/Input
//     PlcTask Inputs/GVL_Devices.MRCO_ROUGH_VRC_04.i_xOpnLS <-> Channel 3/Input
//   plc_mrco_vac Instance <-> Device 1 (EtherCAT)/MRCO_PLC_E00_EK1200/MRCO_PLC_E13_EK1122/MRCO_DRL_03 (EK1100)/MRCO_DRL_03_E02_EL2004
//     PlcTask Outputs/GVL_Devices.MRCO_MSC_VRC_01.q_xOPN_DO <-> Channel 1/Output
//     PlcTask Outputs/GVL_Devices.MRCO_ROUGH_VRC_04.q_xOPN_DO <-> Channel 2/Output
//     PlcTask Outputs/GVL_Devices.MRCO_ROUGH_VRC_05.q_xCLS_DO <-> Channel 3/Output
//   plc_mrco_vac Instance <-> Device 1 (EtherCAT)/MRCO_PLC_E00_EK1200/MRCO_PLC_E13_EK1122/MRCO_DRL_03 (EK1100)/MRCO_DRL_03_E03_EL1004
//     PlcTask Inputs/GVL_Devices.MRCO_ROUGH_VRC_05.i_xClsLS <-> Channel 2/Input
//     PlcTask Inputs/GVL_Devices.MRCO_ROUGH_VRC_05.i_xOpnLS <-> Channel 1/Input
//   plc_mrco_vac Instance <-> Device 1 (EtherCAT)/MRCO_PLC_E00_EK1200/MRCO_PLC_E13_EK1122/MRCO_DRL_03 (EK1100)/MRCO_DRL_03_E04_EL1004
//     PlcTask Inputs/GVL_Devices.MRCO_MSC_PTM_01.i_xAtSpd <-> Channel 2/Input
//     PlcTask Inputs/GVL_Devices.MRCO_MSC_PTM_01.i_xFaultNC <-> Channel 1/Input
//   plc_mrco_vac Instance <-> Device 1 (EtherCAT)/MRCO_PLC_E00_EK1200/MRCO_PLC_E13_EK1122/MRCO_DRL_03 (EK1100)/MRCO_DRL_03_E05_EL6001
//     ComTask Inputs/GVL_COM.stComIn_MRCO_MSC_PTM_01/D[0] <-> COM Inputs/Data In 0
//     ComTask Inputs/GVL_COM.stComIn_MRCO_MSC_PTM_01/D[10] <-> COM Inputs/Data In 10
//     ComTask Inputs/GVL_COM.stComIn_MRCO_MSC_PTM_01/D[11] <-> COM Inputs/Data In 11
//     ComTask Inputs/GVL_COM.stComIn_MRCO_MSC_PTM_01/D[12] <-> COM Inputs/Data In 12
//     ComTask Inputs/GVL_COM.stComIn_MRCO_MSC_PTM_01/D[13] <-> COM Inputs/Data In 13
//     ComTask Inputs/GVL_COM.stComIn_MRCO_MSC_PTM_01/D[14] <-> COM Inputs/Data In 14
//     ComTask Inputs/GVL_COM.stComIn_MRCO_MSC_PTM_01/D[15] <-> COM Inputs/Data In 15
//     ComTask Inputs/GVL_COM.stComIn_MRCO_MSC_PTM_01/D[16] <-> COM Inputs/Data In 16
//     ComTask Inputs/GVL_COM.stComIn_MRCO_MSC_PTM_01/D[17] <-> COM Inputs/Data In 17
//     ComTask Inputs/GVL_COM.stComIn_MRCO_MSC_PTM_01/D[18] <-> COM Inputs/Data In 18
//     ComTask Inputs/GVL_COM.stComIn_MRCO_MSC_PTM_01/D[19] <-> COM Inputs/Data In 19
//     ComTask Inputs/GVL_COM.stComIn_MRCO_MSC_PTM_01/D[1] <-> COM Inputs/Data In 1
//     ComTask Inputs/GVL_COM.stComIn_MRCO_MSC_PTM_01/D[20] <-> COM Inputs/Data In 20
//     ComTask Inputs/GVL_COM.stComIn_MRCO_MSC_PTM_01/D[21] <-> COM Inputs/Data In 21
//     ComTask Inputs/GVL_COM.stComIn_MRCO_MSC_PTM_01/D[2] <-> COM Inputs/Data In 2
//     ComTask Inputs/GVL_COM.stComIn_MRCO_MSC_PTM_01/D[3] <-> COM Inputs/Data In 3
//     ComTask Inputs/GVL_COM.stComIn_MRCO_MSC_PTM_01/D[4] <-> COM Inputs/Data In 4
//     ComTask Inputs/GVL_COM.stComIn_MRCO_MSC_PTM_01/D[5] <-> COM Inputs/Data In 5
//     ComTask Inputs/GVL_COM.stComIn_MRCO_MSC_PTM_01/D[6] <-> COM Inputs/Data In 6
//     ComTask Inputs/GVL_COM.stComIn_MRCO_MSC_PTM_01/D[7] <-> COM Inputs/Data In 7
//     ComTask Inputs/GVL_COM.stComIn_MRCO_MSC_PTM_01/D[8] <-> COM Inputs/Data In 8
//     ComTask Inputs/GVL_COM.stComIn_MRCO_MSC_PTM_01/D[9] <-> COM Inputs/Data In 9
//     ComTask Inputs/GVL_COM.stComIn_MRCO_MSC_PTM_01/Status <-> COM Inputs/Status
//     ComTask Outputs/GVL_COM.stComOut_MRCO_MSC_PTM_01/Ctrl <-> COM Outputs/Ctrl
//     ComTask Outputs/GVL_COM.stComOut_MRCO_MSC_PTM_01/D[0] <-> COM Outputs/Data Out 0
//     ComTask Outputs/GVL_COM.stComOut_MRCO_MSC_PTM_01/D[10] <-> COM Outputs/Data Out 10
//     ComTask Outputs/GVL_COM.stComOut_MRCO_MSC_PTM_01/D[11] <-> COM Outputs/Data Out 11
//     ComTask Outputs/GVL_COM.stComOut_MRCO_MSC_PTM_01/D[12] <-> COM Outputs/Data Out 12
//     ComTask Outputs/GVL_COM.stComOut_MRCO_MSC_PTM_01/D[13] <-> COM Outputs/Data Out 13
//     ComTask Outputs/GVL_COM.stComOut_MRCO_MSC_PTM_01/D[14] <-> COM Outputs/Data Out 14
//     ComTask Outputs/GVL_COM.stComOut_MRCO_MSC_PTM_01/D[15] <-> COM Outputs/Data Out 15
//     ComTask Outputs/GVL_COM.stComOut_MRCO_MSC_PTM_01/D[16] <-> COM Outputs/Data Out 16
//     ComTask Outputs/GVL_COM.stComOut_MRCO_MSC_PTM_01/D[17] <-> COM Outputs/Data Out 17
//     ComTask Outputs/GVL_COM.stComOut_MRCO_MSC_PTM_01/D[18] <-> COM Outputs/Data Out 18
//     ComTask Outputs/GVL_COM.stComOut_MRCO_MSC_PTM_01/D[19] <-> COM Outputs/Data Out 19
//     ComTask Outputs/GVL_COM.stComOut_MRCO_MSC_PTM_01/D[1] <-> COM Outputs/Data Out 1
//     ComTask Outputs/GVL_COM.stComOut_MRCO_MSC_PTM_01/D[20] <-> COM Outputs/Data Out 20
//     ComTask Outputs/GVL_COM.stComOut_MRCO_MSC_PTM_01/D[21] <-> COM Outputs/Data Out 21
//     ComTask Outputs/GVL_COM.stComOut_MRCO_MSC_PTM_01/D[2] <-> COM Outputs/Data Out 2
//     ComTask Outputs/GVL_COM.stComOut_MRCO_MSC_PTM_01/D[3] <-> COM Outputs/Data Out 3
//     ComTask Outputs/GVL_COM.stComOut_MRCO_MSC_PTM_01/D[4] <-> COM Outputs/Data Out 4
//     ComTask Outputs/GVL_COM.stComOut_MRCO_MSC_PTM_01/D[5] <-> COM Outputs/Data Out 5
//     ComTask Outputs/GVL_COM.stComOut_MRCO_MSC_PTM_01/D[6] <-> COM Outputs/Data Out 6
//     ComTask Outputs/GVL_COM.stComOut_MRCO_MSC_PTM_01/D[7] <-> COM Outputs/Data Out 7
//     ComTask Outputs/GVL_COM.stComOut_MRCO_MSC_PTM_01/D[8] <-> COM Outputs/Data Out 8
//     ComTask Outputs/GVL_COM.stComOut_MRCO_MSC_PTM_01/D[9] <-> COM Outputs/Data Out 9
//   plc_mrco_vac Instance <-> Device 1 (EtherCAT)/MRCO_PLC_E00_EK1200/MRCO_PLC_E13_EK1122/MRCO_DRL_03 (EK1100)/MRCO_DRL_03_E06_EL2794
//     PlcTask Outputs/GVL_Devices.MRCO_MSC_GHC_01.q_xHV_DIS <-> Channel 2/Output
//     PlcTask Outputs/GVL_Devices.MRCO_MSC_PTM_01.q_RunDO <-> Channel 1/Output
//   plc_mrco_vac Instance <-> Device 1 (EtherCAT)/MRCO_PLC_E00_EK1200/MRCO_PLC_E13_EK1122/MRCO_DRL_03 (EK1100)/MRCO_DRL_03_E07_EL1084
//     PlcTask Inputs/GVL_Devices.MRCO_MSC_GHC_01.i_xHV_ON <-> Channel 1/Input
//   plc_mrco_vac Instance <-> Device 1 (EtherCAT)/MRCO_PLC_E00_EK1200/MRCO_PLC_E13_EK1122/MRCO_DRL_03 (EK1100)/MRCO_DRL_03_E10_EL3174-0002
//     PlcTask Inputs/GVL_Devices.MRCO_MSC_GHC_01.i_iPRESS_R <-> AI Standard Channel 1/Value
//     PlcTask Inputs/GVL_Devices.MRCO_ROUGH_GPI_05.i_iPRESS_R <-> AI Standard Channel 2/Value
//   plc_mrco_vac Instance <-> Device 1 (EtherCAT)/MRCO_PLC_E00_EK1200/MRCO_PLC_E13_EK1122/MRCO_PNL1_EP01_EP2338-0002
//     PlcTask Inputs/GVL_Devices.MRCO_ROUGH_PTM_01.i_xAtSpd <-> Channel 1/Input
//     PlcTask Inputs/GVL_Devices.MRCO_ROUGH_PTM_01.i_xFaultNC <-> Channel 2/Input
//   plc_mrco_vac Instance <-> Device 1 (EtherCAT)/MRCO_PLC_E00_EK1200/MRCO_PLC_E13_EK1122/MRCO_PNL1_EP02_EP2624-0002
//     PlcTask Outputs/GVL_Devices.MRCO_ROUGH_PTM_01.q_RunDO <-> Channel 1/Output
//     PlcTask Outputs/GVL_Devices.MRCO_ROUGH_PTM_01.q_xReset <-> Channel 2/Output
//   plc_mrco_vac Instance <-> Device 1 (EtherCAT)/MRCO_PLC_E00_EK1200/MRCO_PLC_E13_EK1122/MRCO_PNL1_EP03_EP6002-0002
//     ComTask Inputs/GVL_COM.stComIn_MRCO_ROUGH_PTM_01/D[0] <-> COM TxPDO-Map Inputs Channel 1/Data In 0
//     ComTask Inputs/GVL_COM.stComIn_MRCO_ROUGH_PTM_01/D[10] <-> COM TxPDO-Map Inputs Channel 1/Data In 10
//     ComTask Inputs/GVL_COM.stComIn_MRCO_ROUGH_PTM_01/D[11] <-> COM TxPDO-Map Inputs Channel 1/Data In 11
//     ComTask Inputs/GVL_COM.stComIn_MRCO_ROUGH_PTM_01/D[12] <-> COM TxPDO-Map Inputs Channel 1/Data In 12
//     ComTask Inputs/GVL_COM.stComIn_MRCO_ROUGH_PTM_01/D[13] <-> COM TxPDO-Map Inputs Channel 1/Data In 13
//     ComTask Inputs/GVL_COM.stComIn_MRCO_ROUGH_PTM_01/D[14] <-> COM TxPDO-Map Inputs Channel 1/Data In 14
//     ComTask Inputs/GVL_COM.stComIn_MRCO_ROUGH_PTM_01/D[15] <-> COM TxPDO-Map Inputs Channel 1/Data In 15
//     ComTask Inputs/GVL_COM.stComIn_MRCO_ROUGH_PTM_01/D[16] <-> COM TxPDO-Map Inputs Channel 1/Data In 16
//     ComTask Inputs/GVL_COM.stComIn_MRCO_ROUGH_PTM_01/D[17] <-> COM TxPDO-Map Inputs Channel 1/Data In 17
//     ComTask Inputs/GVL_COM.stComIn_MRCO_ROUGH_PTM_01/D[18] <-> COM TxPDO-Map Inputs Channel 1/Data In 18
//     ComTask Inputs/GVL_COM.stComIn_MRCO_ROUGH_PTM_01/D[19] <-> COM TxPDO-Map Inputs Channel 1/Data In 19
//     ComTask Inputs/GVL_COM.stComIn_MRCO_ROUGH_PTM_01/D[1] <-> COM TxPDO-Map Inputs Channel 1/Data In 1
//     ComTask Inputs/GVL_COM.stComIn_MRCO_ROUGH_PTM_01/D[20] <-> COM TxPDO-Map Inputs Channel 1/Data In 20
//     ComTask Inputs/GVL_COM.stComIn_MRCO_ROUGH_PTM_01/D[21] <-> COM TxPDO-Map Inputs Channel 1/Data In 21
//     ComTask Inputs/GVL_COM.stComIn_MRCO_ROUGH_PTM_01/D[2] <-> COM TxPDO-Map Inputs Channel 1/Data In 2
//     ComTask Inputs/GVL_COM.stComIn_MRCO_ROUGH_PTM_01/D[3] <-> COM TxPDO-Map Inputs Channel 1/Data In 3
//     ComTask Inputs/GVL_COM.stComIn_MRCO_ROUGH_PTM_01/D[4] <-> COM TxPDO-Map Inputs Channel 1/Data In 4
//     ComTask Inputs/GVL_COM.stComIn_MRCO_ROUGH_PTM_01/D[5] <-> COM TxPDO-Map Inputs Channel 1/Data In 5
//     ComTask Inputs/GVL_COM.stComIn_MRCO_ROUGH_PTM_01/D[6] <-> COM TxPDO-Map Inputs Channel 1/Data In 6
//     ComTask Inputs/GVL_COM.stComIn_MRCO_ROUGH_PTM_01/D[7] <-> COM TxPDO-Map Inputs Channel 1/Data In 7
//     ComTask Inputs/GVL_COM.stComIn_MRCO_ROUGH_PTM_01/D[8] <-> COM TxPDO-Map Inputs Channel 1/Data In 8
//     ComTask Inputs/GVL_COM.stComIn_MRCO_ROUGH_PTM_01/D[9] <-> COM TxPDO-Map Inputs Channel 1/Data In 9
//     ComTask Inputs/GVL_COM.stComIn_MRCO_ROUGH_PTM_01/Status <-> COM TxPDO-Map Inputs Channel 1/Status
//     ComTask Outputs/GVL_COM.stComOut_MRCO_ROUGH_PTM_01/Ctrl <-> COM RxPDO-Map Outputs Channel 1/Ctrl
//     ComTask Outputs/GVL_COM.stComOut_MRCO_ROUGH_PTM_01/D[0] <-> COM RxPDO-Map Outputs Channel 1/Data Out 0
//     ComTask Outputs/GVL_COM.stComOut_MRCO_ROUGH_PTM_01/D[10] <-> COM RxPDO-Map Outputs Channel 1/Data Out 10
//     ComTask Outputs/GVL_COM.stComOut_MRCO_ROUGH_PTM_01/D[11] <-> COM RxPDO-Map Outputs Channel 1/Data Out 11
//     ComTask Outputs/GVL_COM.stComOut_MRCO_ROUGH_PTM_01/D[12] <-> COM RxPDO-Map Outputs Channel 1/Data Out 12
//     ComTask Outputs/GVL_COM.stComOut_MRCO_ROUGH_PTM_01/D[13] <-> COM RxPDO-Map Outputs Channel 1/Data Out 13
//     ComTask Outputs/GVL_COM.stComOut_MRCO_ROUGH_PTM_01/D[14] <-> COM RxPDO-Map Outputs Channel 1/Data Out 14
//     ComTask Outputs/GVL_COM.stComOut_MRCO_ROUGH_PTM_01/D[15] <-> COM RxPDO-Map Outputs Channel 1/Data Out 15
//     ComTask Outputs/GVL_COM.stComOut_MRCO_ROUGH_PTM_01/D[16] <-> COM RxPDO-Map Outputs Channel 1/Data Out 16
//     ComTask Outputs/GVL_COM.stComOut_MRCO_ROUGH_PTM_01/D[17] <-> COM RxPDO-Map Outputs Channel 1/Data Out 17
//     ComTask Outputs/GVL_COM.stComOut_MRCO_ROUGH_PTM_01/D[18] <-> COM RxPDO-Map Outputs Channel 1/Data Out 18
//     ComTask Outputs/GVL_COM.stComOut_MRCO_ROUGH_PTM_01/D[19] <-> COM RxPDO-Map Outputs Channel 1/Data Out 19
//     ComTask Outputs/GVL_COM.stComOut_MRCO_ROUGH_PTM_01/D[1] <-> COM RxPDO-Map Outputs Channel 1/Data Out 1
//     ComTask Outputs/GVL_COM.stComOut_MRCO_ROUGH_PTM_01/D[20] <-> COM RxPDO-Map Outputs Channel 1/Data Out 20
//     ComTask Outputs/GVL_COM.stComOut_MRCO_ROUGH_PTM_01/D[21] <-> COM RxPDO-Map Outputs Channel 1/Data Out 21
//     ComTask Outputs/GVL_COM.stComOut_MRCO_ROUGH_PTM_01/D[2] <-> COM RxPDO-Map Outputs Channel 1/Data Out 2
//     ComTask Outputs/GVL_COM.stComOut_MRCO_ROUGH_PTM_01/D[3] <-> COM RxPDO-Map Outputs Channel 1/Data Out 3
//     ComTask Outputs/GVL_COM.stComOut_MRCO_ROUGH_PTM_01/D[4] <-> COM RxPDO-Map Outputs Channel 1/Data Out 4
//     ComTask Outputs/GVL_COM.stComOut_MRCO_ROUGH_PTM_01/D[5] <-> COM RxPDO-Map Outputs Channel 1/Data Out 5
//     ComTask Outputs/GVL_COM.stComOut_MRCO_ROUGH_PTM_01/D[6] <-> COM RxPDO-Map Outputs Channel 1/Data Out 6
//     ComTask Outputs/GVL_COM.stComOut_MRCO_ROUGH_PTM_01/D[7] <-> COM RxPDO-Map Outputs Channel 1/Data Out 7
//     ComTask Outputs/GVL_COM.stComOut_MRCO_ROUGH_PTM_01/D[8] <-> COM RxPDO-Map Outputs Channel 1/Data Out 8
//     ComTask Outputs/GVL_COM.stComOut_MRCO_ROUGH_PTM_01/D[9] <-> COM RxPDO-Map Outputs Channel 1/Data Out 9
//   plc_mrco_vac Instance <-> Device 1 (EtherCAT)/MRCO_PLC_E00_EK1200/MRCO_PLC_E13_EK1122/MRCO_PNL1_EP04_EP3174-0002
//     PlcTask Inputs/GVL_Devices.MRCO_ROUGH_GPI_01.i_iPRESS_R <-> AI Standard Channel 1/Value
//     PlcTask Inputs/GVL_Devices.MRCO_ROUGH_GPI_02.i_iPRESS_R <-> AI Standard Channel 2/Value
//     PlcTask Inputs/GVL_Devices.MRCO_ROUGH_GPI_03.i_iPRESS_R <-> AI Standard Channel 3/Value
//     PlcTask Inputs/GVL_Devices.MRCO_ROUGH_GPI_04.i_iPRESS_R <-> AI Standard Channel 4/Value
//   plc_mrco_vac Instance <-> Device 1 (EtherCAT)/MRCO_PLC_E00_EK1200/MRCO_PLC_E13_EK1122/MRCO_PNL1_EP05_EP3174-0002
//     PlcTask Inputs/GVL_Devices.MRCO_MAIN_GHC_01.i_iPRESS_R <-> AI Standard Channel 2/Value
//     PlcTask Inputs/GVL_Devices.MRCO_MAIN_GPI_01.i_iPRESS_R <-> AI Standard Channel 1/Value
//   plc_mrco_vac Instance <-> Device 1 (EtherCAT)/MRCO_PLC_E00_EK1200/MRCO_PLC_E13_EK1122/MRCO_PNL1_EP06_EP2624-0002
//     PlcTask Outputs/GVL_Devices.MRCO_MAIN_GHC_01.q_xHV_DIS <-> Channel 2/Output
//   plc_mrco_vac Instance <-> Device 1 (EtherCAT)/MRCO_PLC_E00_EK1200/MRCO_PLC_E13_EK1122/MRCO_PNL1_EP07_EP2338-0002
//     PlcTask Inputs/GVL_Devices.MRCO_ROUGH_VRC_01.i_xClsLS <-> Channel 2/Input
//     PlcTask Inputs/GVL_Devices.MRCO_ROUGH_VRC_02.i_xClsLS <-> Channel 6/Input
//     PlcTask Inputs/GVL_Devices.MRCO_ROUGH_VRC_01.i_xOpnLS <-> Channel 1/Input
//     PlcTask Inputs/GVL_Devices.MRCO_ROUGH_VRC_02.i_xOpnLS <-> Channel 5/Input
//     PlcTask Outputs/GVL_Devices.MRCO_ROUGH_VRC_01.q_xOPN_DO <-> Channel 11/Output
//     PlcTask Outputs/GVL_Devices.MRCO_ROUGH_VRC_02.q_xCLS_DO <-> Channel 15/Output
//   plc_mrco_vac Instance <-> Device 1 (EtherCAT)/MRCO_PLC_E00_EK1200/MRCO_PLC_E13_EK1122/MRCO_PNL1_EP08_EP2338-0002
//     PlcTask Inputs/GVL_Devices.MRCO_ROUGH_VRC_03.i_xClsLS <-> Channel 2/Input
//     PlcTask Inputs/GVL_Devices.MRCO_ROUGH_VRC_06.i_xClsLS <-> Channel 6/Input
//     PlcTask Inputs/GVL_Devices.MRCO_ROUGH_VRC_03.i_xOpnLS <-> Channel 1/Input
//     PlcTask Inputs/GVL_Devices.MRCO_ROUGH_VRC_06.i_xOpnLS <-> Channel 5/Input
//     PlcTask Outputs/GVL_Devices.MRCO_ROUGH_VRC_03.q_xOPN_DO <-> Channel 11/Output
//     PlcTask Outputs/GVL_Devices.MRCO_ROUGH_VRC_06.q_xOPN_DO <-> Channel 15/Output
//   plc_mrco_vac Instance <-> Device 1 (EtherCAT)/MRCO_PLC_E00_EK1200/MRCO_PLC_E13_EK1122/VCN_1_VAT590
//     PlcTask Inputs/GVL_Devices.MRCO_VCN_01.i_bValveEthCatStatus <-> WcState/WcState
//     PlcTask Inputs/GVL_Devices.MRCO_VCN_01.i_eControlMode <-> DI TxPDO-Map/Control mode
//     PlcTask Inputs/GVL_Devices.MRCO_VCN_01.i_eFatalError <-> DI TxPDO-Map/Fatal error
//     PlcTask Inputs/GVL_Devices.MRCO_VCN_01.i_nRawPosition <-> DI TxPDO-Map/Position
//     PlcTask Inputs/GVL_Devices.MRCO_VCN_01.i_nRawPressure <-> DI TxPDO-Map/Pressure
//     PlcTask Inputs/GVL_Devices.MRCO_VCN_01.i_stExtnWarnings <-> DI TxPDO-Map/Extended warnings
//     PlcTask Inputs/GVL_Devices.MRCO_VCN_01.i_stGenStatus <-> DI TxPDO-Map/General status
//     PlcTask Inputs/GVL_Devices.MRCO_VCN_01.i_stGenWarnings <-> DI TxPDO-Map/General warnings
//     PlcTask Inputs/GVL_Devices.MRCO_VCN_01.i_stVat590PlcDriveRef/aNetId <-> InfoData/AdsAddr/netId
//     PlcTask Inputs/GVL_Devices.MRCO_VCN_01.i_stVat590PlcDriveRef/nSlaveAddr <-> InfoData/AdsAddr/port
//     PlcTask Outputs/GVL_Devices.MRCO_VCN_01.o_eCtrlModeSP <-> DO RxPDO-Map/Control mode setpoint
//     PlcTask Outputs/GVL_Devices.MRCO_VCN_01.o_nRawPositionSP <-> DO RxPDO-Map/Position setpoint
//     PlcTask Outputs/GVL_Devices.MRCO_VCN_01.o_nRawPressure <-> DO RxPDO-Map/External digital pressure sensor 1
//     PlcTask Outputs/GVL_Devices.MRCO_VCN_01.o_nRawPressureSP <-> DO RxPDO-Map/Pressure setpoint
//     PlcTask Outputs/GVL_Devices.MRCO_VCN_01.o_stGenCtrlSP <-> DO RxPDO-Map/General control setpoint

CONFIGURATION plc_mrco_vac
    RESOURCE PLC ON TwinCAT3
        TASK ComTask(INTERVAL := T#10ms, PRIORITY := 15);
        TASK PlcTask(INTERVAL := T#10ms, PRIORITY := 20);
        PROGRAM PRG_COM WITH ComTask : PRG_COM;
        PROGRAM MAIN WITH PlcTask : MAIN;
    END_RESOURCE
END_CONFIGURATION

// ---- GVLs/GVL_COM.TcGVL
//{attribute 'qualified_only'}
VAR_GLOBAL
    // Define COM Ports/Buffers incl. library Tc2_SerialCom
    SerialRXBuffer_MRCO_MAIN_PTM_01 : ComBuffer;
    SerialTXBuffer_MRCO_MAIN_PTM_01 : ComBuffer;
    SerialRXBuffer_MRCO_MAIN_PTM_02 : ComBuffer;
    SerialTXBuffer_MRCO_MAIN_PTM_02 : ComBuffer;
    SerialRXBuffer_MRCO_MAIN_PTM_03 : ComBuffer;
    SerialTXBuffer_MRCO_MAIN_PTM_03 : ComBuffer;
    SerialRXBuffer_MRCO_MAIN_PTM_04 : ComBuffer;
    SerialTXBuffer_MRCO_MAIN_PTM_04 : ComBuffer;
    SerialRXBuffer_MRCO_ROUGH_PTM_01 : ComBuffer;
    SerialTXBuffer_MRCO_ROUGH_PTM_01 : ComBuffer;
    SerialRXBuffer_MRCO_MSC_PTM_01 : ComBuffer;
    SerialTXBuffer_MRCO_MSC_PTM_01 : ComBuffer;


    // Serial Terminal
    fbSerialLineControl_MRCO_MAIN_PTM_01 : SerialLineControl;
    fbSerialLineControl_MRCO_MAIN_PTM_02 : SerialLineControl;
    fbSerialLineControl_MRCO_MAIN_PTM_03 : SerialLineControl;
    fbSerialLineControl_MRCO_MAIN_PTM_04 : SerialLineControl;
    fbSerialLineControl_MRCO_ROUGH_PTM_01 : SerialLineControl;
    fbSerialLineControl_MRCO_MSC_PTM_01 : SerialLineControl;


    //SERIAL IO
    {attribute      'TcLinkTo'      :=      '.Status:=TIIB[MRCO_PLC_E11_EL6002]^COM TxPDO-Map Inputs Channel 1^Status;
                                                            .D[0]:=TIIB[MRCO_PLC_E11_EL6002]^COM TxPDO-Map Inputs Channel 1^Data In 0;
                                                            .D[1]:=TIIB[MRCO_PLC_E11_EL6002]^COM TxPDO-Map Inputs Channel 1^Data In 1;
                                                            .D[2]:=TIIB[MRCO_PLC_E11_EL6002]^COM TxPDO-Map Inputs Channel 1^Data In 2;
                                                            .D[3]:=TIIB[MRCO_PLC_E11_EL6002]^COM TxPDO-Map Inputs Channel 1^Data In 3;
                                                            .D[4]:=TIIB[MRCO_PLC_E11_EL6002]^COM TxPDO-Map Inputs Channel 1^Data In 4;
                                                            .D[5]:=TIIB[MRCO_PLC_E11_EL6002]^COM TxPDO-Map Inputs Channel 1^Data In 5;
                                                            .D[6]:=TIIB[MRCO_PLC_E11_EL6002]^COM TxPDO-Map Inputs Channel 1^Data In 6;
                                                            .D[7]:=TIIB[MRCO_PLC_E11_EL6002]^COM TxPDO-Map Inputs Channel 1^Data In 7;
                                                            .D[8]:=TIIB[MRCO_PLC_E11_EL6002]^COM TxPDO-Map Inputs Channel 1^Data In 8;
                                                            .D[9]:=TIIB[MRCO_PLC_E11_EL6002]^COM TxPDO-Map Inputs Channel 1^Data In 9;
                                                            .D[10]:=TIIB[MRCO_PLC_E11_EL6002]^COM TxPDO-Map Inputs Channel 1^Data In 10;
                                                            .D[11]:=TIIB[MRCO_PLC_E11_EL6002]^COM TxPDO-Map Inputs Channel 1^Data In 11;
                                                            .D[12]:=TIIB[MRCO_PLC_E11_EL6002]^COM TxPDO-Map Inputs Channel 1^Data In 12;
                                                            .D[13]:=TIIB[MRCO_PLC_E11_EL6002]^COM TxPDO-Map Inputs Channel 1^Data In 13;
                                                            .D[14]:=TIIB[MRCO_PLC_E11_EL6002]^COM TxPDO-Map Inputs Channel 1^Data In 14;
                                                            .D[15]:=TIIB[MRCO_PLC_E11_EL6002]^COM TxPDO-Map Inputs Channel 1^Data In 15;
                                                            .D[16]:=TIIB[MRCO_PLC_E11_EL6002]^COM TxPDO-Map Inputs Channel 1^Data In 16;
                                                            .D[17]:=TIIB[MRCO_PLC_E11_EL6002]^COM TxPDO-Map Inputs Channel 1^Data In 17;
                                                            .D[18]:=TIIB[MRCO_PLC_E11_EL6002]^COM TxPDO-Map Inputs Channel 1^Data In 18;
                                                            .D[19]:=TIIB[MRCO_PLC_E11_EL6002]^COM TxPDO-Map Inputs Channel 1^Data In 19;
                                                            .D[20]:=TIIB[MRCO_PLC_E11_EL6002]^COM TxPDO-Map Inputs Channel 1^Data In 20;
                                                            .D[21]:=TIIB[MRCO_PLC_E11_EL6002]^COM TxPDO-Map Inputs Channel 1^Data In 21
    '}
    stComIn_MRCO_MAIN_PTM_01        AT %I*  :       EL6inData22B;

    {attribute      'TcLinkTo'      :=      '.Ctrl:=TIIB[MRCO_PLC_E11_EL6002]^COM RxPDO-Map Outputs Channel 1^Ctrl;
                                                            .D[0]:=TIIB[MRCO_PLC_E11_EL6002]^COM RxPDO-Map Outputs Channel 1^Data Out 0;
                                                            .D[1]:=TIIB[MRCO_PLC_E11_EL6002]^COM RxPDO-Map Outputs Channel 1^Data Out 1;
                                                            .D[2]:=TIIB[MRCO_PLC_E11_EL6002]^COM RxPDO-Map Outputs Channel 1^Data Out 2;
                                                            .D[3]:=TIIB[MRCO_PLC_E11_EL6002]^COM RxPDO-Map Outputs Channel 1^Data Out 3;
                                                            .D[4]:=TIIB[MRCO_PLC_E11_EL6002]^COM RxPDO-Map Outputs Channel 1^Data Out 4;
                                                            .D[5]:=TIIB[MRCO_PLC_E11_EL6002]^COM RxPDO-Map Outputs Channel 1^Data Out 5;
                                                            .D[6]:=TIIB[MRCO_PLC_E11_EL6002]^COM RxPDO-Map Outputs Channel 1^Data Out 6;
                                                            .D[7]:=TIIB[MRCO_PLC_E11_EL6002]^COM RxPDO-Map Outputs Channel 1^Data Out 7;
                                                            .D[8]:=TIIB[MRCO_PLC_E11_EL6002]^COM RxPDO-Map Outputs Channel 1^Data Out 8;
                                                            .D[9]:=TIIB[MRCO_PLC_E11_EL6002]^COM RxPDO-Map Outputs Channel 1^Data Out 9;
                                                            .D[10]:=TIIB[MRCO_PLC_E11_EL6002]^COM RxPDO-Map Outputs Channel 1^Data Out 10;
                                                            .D[11]:=TIIB[MRCO_PLC_E11_EL6002]^COM RxPDO-Map Outputs Channel 1^Data Out 11;
                                                            .D[12]:=TIIB[MRCO_PLC_E11_EL6002]^COM RxPDO-Map Outputs Channel 1^Data Out 12;
                                                            .D[13]:=TIIB[MRCO_PLC_E11_EL6002]^COM RxPDO-Map Outputs Channel 1^Data Out 13;
                                                            .D[14]:=TIIB[MRCO_PLC_E11_EL6002]^COM RxPDO-Map Outputs Channel 1^Data Out 14;
                                                            .D[15]:=TIIB[MRCO_PLC_E11_EL6002]^COM RxPDO-Map Outputs Channel 1^Data Out 15;
                                                            .D[16]:=TIIB[MRCO_PLC_E11_EL6002]^COM RxPDO-Map Outputs Channel 1^Data Out 16;
                                                            .D[17]:=TIIB[MRCO_PLC_E11_EL6002]^COM RxPDO-Map Outputs Channel 1^Data Out 17;
                                                            .D[18]:=TIIB[MRCO_PLC_E11_EL6002]^COM RxPDO-Map Outputs Channel 1^Data Out 18;
                                                            .D[19]:=TIIB[MRCO_PLC_E11_EL6002]^COM RxPDO-Map Outputs Channel 1^Data Out 19;
                                                            .D[20]:=TIIB[MRCO_PLC_E11_EL6002]^COM RxPDO-Map Outputs Channel 1^Data Out 20;
                                                            .D[21]:=TIIB[MRCO_PLC_E11_EL6002]^COM RxPDO-Map Outputs Channel 1^Data Out 21
    '}
    stComOut_MRCO_MAIN_PTM_01        AT %Q*  :       EL6outData22B;

    {attribute      'TcLinkTo'      :=      '.Status:=TIIB[MRCO_PLC_E11_EL6002]^COM TxPDO-Map Inputs Channel 2^Status;
                                                            .D[0]:=TIIB[MRCO_PLC_E11_EL6002]^COM TxPDO-Map Inputs Channel 2^Data In 0;
                                                            .D[1]:=TIIB[MRCO_PLC_E11_EL6002]^COM TxPDO-Map Inputs Channel 2^Data In 1;
                                                            .D[2]:=TIIB[MRCO_PLC_E11_EL6002]^COM TxPDO-Map Inputs Channel 2^Data In 2;
                                                            .D[3]:=TIIB[MRCO_PLC_E11_EL6002]^COM TxPDO-Map Inputs Channel 2^Data In 3;
                                                            .D[4]:=TIIB[MRCO_PLC_E11_EL6002]^COM TxPDO-Map Inputs Channel 2^Data In 4;
                                                            .D[5]:=TIIB[MRCO_PLC_E11_EL6002]^COM TxPDO-Map Inputs Channel 2^Data In 5;
                                                            .D[6]:=TIIB[MRCO_PLC_E11_EL6002]^COM TxPDO-Map Inputs Channel 2^Data In 6;
                                                            .D[7]:=TIIB[MRCO_PLC_E11_EL6002]^COM TxPDO-Map Inputs Channel 2^Data In 7;
                                                            .D[8]:=TIIB[MRCO_PLC_E11_EL6002]^COM TxPDO-Map Inputs Channel 2^Data In 8;
                                                            .D[9]:=TIIB[MRCO_PLC_E11_EL6002]^COM TxPDO-Map Inputs Channel 2^Data In 9;
                                                            .D[10]:=TIIB[MRCO_PLC_E11_EL6002]^COM TxPDO-Map Inputs Channel 2^Data In 10;
                                                            .D[11]:=TIIB[MRCO_PLC_E11_EL6002]^COM TxPDO-Map Inputs Channel 2^Data In 11;
                                                            .D[12]:=TIIB[MRCO_PLC_E11_EL6002]^COM TxPDO-Map Inputs Channel 2^Data In 12;
                                                            .D[13]:=TIIB[MRCO_PLC_E11_EL6002]^COM TxPDO-Map Inputs Channel 2^Data In 13;
                                                            .D[14]:=TIIB[MRCO_PLC_E11_EL6002]^COM TxPDO-Map Inputs Channel 2^Data In 14;
                                                            .D[15]:=TIIB[MRCO_PLC_E11_EL6002]^COM TxPDO-Map Inputs Channel 2^Data In 15;
                                                            .D[16]:=TIIB[MRCO_PLC_E11_EL6002]^COM TxPDO-Map Inputs Channel 2^Data In 16;
                                                            .D[17]:=TIIB[MRCO_PLC_E11_EL6002]^COM TxPDO-Map Inputs Channel 2^Data In 17;
                                                            .D[18]:=TIIB[MRCO_PLC_E11_EL6002]^COM TxPDO-Map Inputs Channel 2^Data In 18;
                                                            .D[19]:=TIIB[MRCO_PLC_E11_EL6002]^COM TxPDO-Map Inputs Channel 2^Data In 19;
                                                            .D[20]:=TIIB[MRCO_PLC_E11_EL6002]^COM TxPDO-Map Inputs Channel 2^Data In 20;
                                                            .D[21]:=TIIB[MRCO_PLC_E11_EL6002]^COM TxPDO-Map Inputs Channel 2^Data In 21
    '}
    stComIn_MRCO_MAIN_PTM_03        AT %I*  :       EL6inData22B;

    {attribute      'TcLinkTo'      :=      '.Ctrl:=TIIB[MRCO_PLC_E11_EL6002]^COM RxPDO-Map Outputs Channel 2^Ctrl;
                                                            .D[0]:=TIIB[MRCO_PLC_E11_EL6002]^COM RxPDO-Map Outputs Channel 2^Data Out 0;
                                                            .D[1]:=TIIB[MRCO_PLC_E11_EL6002]^COM RxPDO-Map Outputs Channel 2^Data Out 1;
                                                            .D[2]:=TIIB[MRCO_PLC_E11_EL6002]^COM RxPDO-Map Outputs Channel 2^Data Out 2;
                                                            .D[3]:=TIIB[MRCO_PLC_E11_EL6002]^COM RxPDO-Map Outputs Channel 2^Data Out 3;
                                                            .D[4]:=TIIB[MRCO_PLC_E11_EL6002]^COM RxPDO-Map Outputs Channel 2^Data Out 4;
                                                            .D[5]:=TIIB[MRCO_PLC_E11_EL6002]^COM RxPDO-Map Outputs Channel 2^Data Out 5;
                                                            .D[6]:=TIIB[MRCO_PLC_E11_EL6002]^COM RxPDO-Map Outputs Channel 2^Data Out 6;
                                                            .D[7]:=TIIB[MRCO_PLC_E11_EL6002]^COM RxPDO-Map Outputs Channel 2^Data Out 7;
                                                            .D[8]:=TIIB[MRCO_PLC_E11_EL6002]^COM RxPDO-Map Outputs Channel 2^Data Out 8;
                                                            .D[9]:=TIIB[MRCO_PLC_E11_EL6002]^COM RxPDO-Map Outputs Channel 2^Data Out 9;
                                                            .D[10]:=TIIB[MRCO_PLC_E11_EL6002]^COM RxPDO-Map Outputs Channel 2^Data Out 10;
                                                            .D[11]:=TIIB[MRCO_PLC_E11_EL6002]^COM RxPDO-Map Outputs Channel 2^Data Out 11;
                                                            .D[12]:=TIIB[MRCO_PLC_E11_EL6002]^COM RxPDO-Map Outputs Channel 2^Data Out 12;
                                                            .D[13]:=TIIB[MRCO_PLC_E11_EL6002]^COM RxPDO-Map Outputs Channel 2^Data Out 13;
                                                            .D[14]:=TIIB[MRCO_PLC_E11_EL6002]^COM RxPDO-Map Outputs Channel 2^Data Out 14;
                                                            .D[15]:=TIIB[MRCO_PLC_E11_EL6002]^COM RxPDO-Map Outputs Channel 2^Data Out 15;
                                                            .D[16]:=TIIB[MRCO_PLC_E11_EL6002]^COM RxPDO-Map Outputs Channel 2^Data Out 16;
                                                            .D[17]:=TIIB[MRCO_PLC_E11_EL6002]^COM RxPDO-Map Outputs Channel 2^Data Out 17;
                                                            .D[18]:=TIIB[MRCO_PLC_E11_EL6002]^COM RxPDO-Map Outputs Channel 2^Data Out 18;
                                                            .D[19]:=TIIB[MRCO_PLC_E11_EL6002]^COM RxPDO-Map Outputs Channel 2^Data Out 19;
                                                            .D[20]:=TIIB[MRCO_PLC_E11_EL6002]^COM RxPDO-Map Outputs Channel 2^Data Out 20;
                                                            .D[21]:=TIIB[MRCO_PLC_E11_EL6002]^COM RxPDO-Map Outputs Channel 2^Data Out 21
    '}
    stComOut_MRCO_MAIN_PTM_03        AT %Q*  :       EL6outData22B;

    {attribute      'TcLinkTo'      :=      '.Status:=TIIB[MRCO_PLC_E12_EL6002]^COM TxPDO-Map Inputs Channel 1^Status;
                                                            .D[0]:=TIIB[MRCO_PLC_E12_EL6002]^COM TxPDO-Map Inputs Channel 1^Data In 0;
                                                            .D[1]:=TIIB[MRCO_PLC_E12_EL6002]^COM TxPDO-Map Inputs Channel 1^Data In 1;
                                                            .D[2]:=TIIB[MRCO_PLC_E12_EL6002]^COM TxPDO-Map Inputs Channel 1^Data In 2;
                                                            .D[3]:=TIIB[MRCO_PLC_E12_EL6002]^COM TxPDO-Map Inputs Channel 1^Data In 3;
                                                            .D[4]:=TIIB[MRCO_PLC_E12_EL6002]^COM TxPDO-Map Inputs Channel 1^Data In 4;
                                                            .D[5]:=TIIB[MRCO_PLC_E12_EL6002]^COM TxPDO-Map Inputs Channel 1^Data In 5;
                                                            .D[6]:=TIIB[MRCO_PLC_E12_EL6002]^COM TxPDO-Map Inputs Channel 1^Data In 6;
                                                            .D[7]:=TIIB[MRCO_PLC_E12_EL6002]^COM TxPDO-Map Inputs Channel 1^Data In 7;
                                                            .D[8]:=TIIB[MRCO_PLC_E12_EL6002]^COM TxPDO-Map Inputs Channel 1^Data In 8;
                                                            .D[9]:=TIIB[MRCO_PLC_E12_EL6002]^COM TxPDO-Map Inputs Channel 1^Data In 9;
                                                            .D[10]:=TIIB[MRCO_PLC_E12_EL6002]^COM TxPDO-Map Inputs Channel 1^Data In 10;
                                                            .D[11]:=TIIB[MRCO_PLC_E12_EL6002]^COM TxPDO-Map Inputs Channel 1^Data In 11;
                                                            .D[12]:=TIIB[MRCO_PLC_E12_EL6002]^COM TxPDO-Map Inputs Channel 1^Data In 12;
                                                            .D[13]:=TIIB[MRCO_PLC_E12_EL6002]^COM TxPDO-Map Inputs Channel 1^Data In 13;
                                                            .D[14]:=TIIB[MRCO_PLC_E12_EL6002]^COM TxPDO-Map Inputs Channel 1^Data In 14;
                                                            .D[15]:=TIIB[MRCO_PLC_E12_EL6002]^COM TxPDO-Map Inputs Channel 1^Data In 15;
                                                            .D[16]:=TIIB[MRCO_PLC_E12_EL6002]^COM TxPDO-Map Inputs Channel 1^Data In 16;
                                                            .D[17]:=TIIB[MRCO_PLC_E12_EL6002]^COM TxPDO-Map Inputs Channel 1^Data In 17;
                                                            .D[18]:=TIIB[MRCO_PLC_E12_EL6002]^COM TxPDO-Map Inputs Channel 1^Data In 18;
                                                            .D[19]:=TIIB[MRCO_PLC_E12_EL6002]^COM TxPDO-Map Inputs Channel 1^Data In 19;
                                                            .D[20]:=TIIB[MRCO_PLC_E12_EL6002]^COM TxPDO-Map Inputs Channel 1^Data In 20;
                                                            .D[21]:=TIIB[MRCO_PLC_E12_EL6002]^COM TxPDO-Map Inputs Channel 1^Data In 21
    '}
    stComIn_MRCO_MAIN_PTM_02        AT %I*  :       EL6inData22B;

    {attribute      'TcLinkTo'      :=      '.Ctrl:=TIIB[MRCO_PLC_E12_EL6002]^COM RxPDO-Map Outputs Channel 1^Ctrl;=
                                                            .D[0]:=TIIB[MRCO_PLC_E12_EL6002]^COM RxPDO-Map Outputs Channel 1^Data Out 0;
                                                            .D[1]:=TIIB[MRCO_PLC_E12_EL6002]^COM RxPDO-Map Outputs Channel 1^Data Out 1;
                                                            .D[2]:=TIIB[MRCO_PLC_E12_EL6002]^COM RxPDO-Map Outputs Channel 1^Data Out 2;
                                                            .D[3]:=TIIB[MRCO_PLC_E12_EL6002]^COM RxPDO-Map Outputs Channel 1^Data Out 3;
                                                            .D[4]:=TIIB[MRCO_PLC_E12_EL6002]^COM RxPDO-Map Outputs Channel 1^Data Out 4;
                                                            .D[5]:=TIIB[MRCO_PLC_E12_EL6002]^COM RxPDO-Map Outputs Channel 1^Data Out 5;
                                                            .D[6]:=TIIB[MRCO_PLC_E12_EL6002]^COM RxPDO-Map Outputs Channel 1^Data Out 6;
                                                            .D[7]:=TIIB[MRCO_PLC_E12_EL6002]^COM RxPDO-Map Outputs Channel 1^Data Out 7;
                                                            .D[8]:=TIIB[MRCO_PLC_E12_EL6002]^COM RxPDO-Map Outputs Channel 1^Data Out 8;
                                                            .D[9]:=TIIB[MRCO_PLC_E12_EL6002]^COM RxPDO-Map Outputs Channel 1^Data Out 9;
                                                            .D[10]:=TIIB[MRCO_PLC_E12_EL6002]^COM RxPDO-Map Outputs Channel 1^Data Out 10;
                                                            .D[11]:=TIIB[MRCO_PLC_E12_EL6002]^COM RxPDO-Map Outputs Channel 1^Data Out 11;
                                                            .D[12]:=TIIB[MRCO_PLC_E12_EL6002]^COM RxPDO-Map Outputs Channel 1^Data Out 12;
                                                            .D[13]:=TIIB[MRCO_PLC_E12_EL6002]^COM RxPDO-Map Outputs Channel 1^Data Out 13;
                                                            .D[14]:=TIIB[MRCO_PLC_E12_EL6002]^COM RxPDO-Map Outputs Channel 1^Data Out 14;
                                                            .D[15]:=TIIB[MRCO_PLC_E12_EL6002]^COM RxPDO-Map Outputs Channel 1^Data Out 15;
                                                            .D[16]:=TIIB[MRCO_PLC_E12_EL6002]^COM RxPDO-Map Outputs Channel 1^Data Out 16;
                                                            .D[17]:=TIIB[MRCO_PLC_E12_EL6002]^COM RxPDO-Map Outputs Channel 1^Data Out 17;
                                                            .D[18]:=TIIB[MRCO_PLC_E12_EL6002]^COM RxPDO-Map Outputs Channel 1^Data Out 18;
                                                            .D[19]:=TIIB[MRCO_PLC_E12_EL6002]^COM RxPDO-Map Outputs Channel 1^Data Out 19;
                                                            .D[20]:=TIIB[MRCO_PLC_E12_EL6002]^COM RxPDO-Map Outputs Channel 1^Data Out 20;
                                                            .D[21]:=TIIB[MRCO_PLC_E12_EL6002]^COM RxPDO-Map Outputs Channel 1^Data Out 21
    '}
    stComOut_MRCO_MAIN_PTM_02        AT %Q*  :       EL6outData22B;

    {attribute      'TcLinkTo'      :=      '.Status:=TIIB[MRCO_PLC_E12_EL6002]^COM TxPDO-Map Inputs Channel 2^Status;
                                                            .D[0]:=TIIB[MRCO_PLC_E12_EL6002]^COM TxPDO-Map Inputs Channel 2^Data In 0;
                                                            .D[1]:=TIIB[MRCO_PLC_E12_EL6002]^COM TxPDO-Map Inputs Channel 2^Data In 1;
                                                            .D[2]:=TIIB[MRCO_PLC_E12_EL6002]^COM TxPDO-Map Inputs Channel 2^Data In 2;
                                                            .D[3]:=TIIB[MRCO_PLC_E12_EL6002]^COM TxPDO-Map Inputs Channel 2^Data In 3;
                                                            .D[4]:=TIIB[MRCO_PLC_E12_EL6002]^COM TxPDO-Map Inputs Channel 2^Data In 4;
                                                            .D[5]:=TIIB[MRCO_PLC_E12_EL6002]^COM TxPDO-Map Inputs Channel 2^Data In 5;
                                                            .D[6]:=TIIB[MRCO_PLC_E12_EL6002]^COM TxPDO-Map Inputs Channel 2^Data In 6;
                                                            .D[7]:=TIIB[MRCO_PLC_E12_EL6002]^COM TxPDO-Map Inputs Channel 2^Data In 7;
                                                            .D[8]:=TIIB[MRCO_PLC_E12_EL6002]^COM TxPDO-Map Inputs Channel 2^Data In 8;
                                                            .D[9]:=TIIB[MRCO_PLC_E12_EL6002]^COM TxPDO-Map Inputs Channel 2^Data In 9;
                                                            .D[10]:=TIIB[MRCO_PLC_E12_EL6002]^COM TxPDO-Map Inputs Channel 2^Data In 10;
                                                            .D[11]:=TIIB[MRCO_PLC_E12_EL6002]^COM TxPDO-Map Inputs Channel 2^Data In 11;
                                                            .D[12]:=TIIB[MRCO_PLC_E12_EL6002]^COM TxPDO-Map Inputs Channel 2^Data In 12;
                                                            .D[13]:=TIIB[MRCO_PLC_E12_EL6002]^COM TxPDO-Map Inputs Channel 2^Data In 13;
                                                            .D[14]:=TIIB[MRCO_PLC_E12_EL6002]^COM TxPDO-Map Inputs Channel 2^Data In 14;
                                                            .D[15]:=TIIB[MRCO_PLC_E12_EL6002]^COM TxPDO-Map Inputs Channel 2^Data In 15;
                                                            .D[16]:=TIIB[MRCO_PLC_E12_EL6002]^COM TxPDO-Map Inputs Channel 2^Data In 16;
                                                            .D[17]:=TIIB[MRCO_PLC_E12_EL6002]^COM TxPDO-Map Inputs Channel 2^Data In 17;
                                                            .D[18]:=TIIB[MRCO_PLC_E12_EL6002]^COM TxPDO-Map Inputs Channel 2^Data In 18;
                                                            .D[19]:=TIIB[MRCO_PLC_E12_EL6002]^COM TxPDO-Map Inputs Channel 2^Data In 19;
                                                            .D[20]:=TIIB[MRCO_PLC_E12_EL6002]^COM TxPDO-Map Inputs Channel 2^Data In 20;
                                                            .D[21]:=TIIB[MRCO_PLC_E12_EL6002]^COM TxPDO-Map Inputs Channel 2^Data In 21
    '}
    stComIn_MRCO_MAIN_PTM_04        AT %I*  :       EL6inData22B;

    {attribute      'TcLinkTo'      :=      '.Ctrl:=TIIB[MRCO_PLC_E12_EL6002]^COM RxPDO-Map Outputs Channel 2^Ctrl;
                                                            .D[0]:=TIIB[MRCO_PLC_E12_EL6002]^COM RxPDO-Map Outputs Channel 2^Data Out 0;
                                                            .D[1]:=TIIB[MRCO_PLC_E12_EL6002]^COM RxPDO-Map Outputs Channel 2^Data Out 1;
                                                            .D[2]:=TIIB[MRCO_PLC_E12_EL6002]^COM RxPDO-Map Outputs Channel 2^Data Out 2;
                                                            .D[3]:=TIIB[MRCO_PLC_E12_EL6002]^COM RxPDO-Map Outputs Channel 2^Data Out 3;
                                                            .D[4]:=TIIB[MRCO_PLC_E12_EL6002]^COM RxPDO-Map Outputs Channel 2^Data Out 4;
                                                            .D[5]:=TIIB[MRCO_PLC_E12_EL6002]^COM RxPDO-Map Outputs Channel 2^Data Out 5;
                                                            .D[6]:=TIIB[MRCO_PLC_E12_EL6002]^COM RxPDO-Map Outputs Channel 2^Data Out 6;
                                                            .D[7]:=TIIB[MRCO_PLC_E12_EL6002]^COM RxPDO-Map Outputs Channel 2^Data Out 7;
                                                            .D[8]:=TIIB[MRCO_PLC_E12_EL6002]^COM RxPDO-Map Outputs Channel 2^Data Out 8;
                                                            .D[9]:=TIIB[MRCO_PLC_E12_EL6002]^COM RxPDO-Map Outputs Channel 2^Data Out 9;
                                                            .D[10]:=TIIB[MRCO_PLC_E12_EL6002]^COM RxPDO-Map Outputs Channel 2^Data Out 10;
                                                            .D[11]:=TIIB[MRCO_PLC_E12_EL6002]^COM RxPDO-Map Outputs Channel 2^Data Out 11;
                                                            .D[12]:=TIIB[MRCO_PLC_E12_EL6002]^COM RxPDO-Map Outputs Channel 2^Data Out 12;
                                                            .D[13]:=TIIB[MRCO_PLC_E12_EL6002]^COM RxPDO-Map Outputs Channel 2^Data Out 13;
                                                            .D[14]:=TIIB[MRCO_PLC_E12_EL6002]^COM RxPDO-Map Outputs Channel 2^Data Out 14;
                                                            .D[15]:=TIIB[MRCO_PLC_E12_EL6002]^COM RxPDO-Map Outputs Channel 2^Data Out 15;
                                                            .D[16]:=TIIB[MRCO_PLC_E12_EL6002]^COM RxPDO-Map Outputs Channel 2^Data Out 16;
                                                            .D[17]:=TIIB[MRCO_PLC_E12_EL6002]^COM RxPDO-Map Outputs Channel 2^Data Out 17;
                                                            .D[18]:=TIIB[MRCO_PLC_E12_EL6002]^COM RxPDO-Map Outputs Channel 2^Data Out 18;
                                                            .D[19]:=TIIB[MRCO_PLC_E12_EL6002]^COM RxPDO-Map Outputs Channel 2^Data Out 19;
                                                            .D[20]:=TIIB[MRCO_PLC_E12_EL6002]^COM RxPDO-Map Outputs Channel 2^Data Out 20;
                                                            .D[21]:=TIIB[MRCO_PLC_E12_EL6002]^COM RxPDO-Map Outputs Channel 2^Data Out 21
    '}
    stComOut_MRCO_MAIN_PTM_04        AT %Q*  :       EL6outData22B;

    {attribute      'TcLinkTo'      :=      '.Status:=TIIB[MRCO_PNL1_EP03_EP6002-0002]^COM TxPDO-Map Inputs Channel 1^Status;
                                                            .D[0]:=TIIB[MRCO_PNL1_EP03_EP6002-0002]^COM TxPDO-Map Inputs Channel 1^Data In 0;
                                                            .D[1]:=TIIB[MRCO_PNL1_EP03_EP6002-0002]^COM TxPDO-Map Inputs Channel 1^Data In 1;
                                                            .D[2]:=TIIB[MRCO_PNL1_EP03_EP6002-0002]^COM TxPDO-Map Inputs Channel 1^Data In 2;
                                                            .D[3]:=TIIB[MRCO_PNL1_EP03_EP6002-0002]^COM TxPDO-Map Inputs Channel 1^Data In 3;
                                                            .D[4]:=TIIB[MRCO_PNL1_EP03_EP6002-0002]^COM TxPDO-Map Inputs Channel 1^Data In 4;
                                                            .D[5]:=TIIB[MRCO_PNL1_EP03_EP6002-0002]^COM TxPDO-Map Inputs Channel 1^Data In 5;
                                                            .D[6]:=TIIB[MRCO_PNL1_EP03_EP6002-0002]^COM TxPDO-Map Inputs Channel 1^Data In 6;
                                                            .D[7]:=TIIB[MRCO_PNL1_EP03_EP6002-0002]^COM TxPDO-Map Inputs Channel 1^Data In 7;
                                                            .D[8]:=TIIB[MRCO_PNL1_EP03_EP6002-0002]^COM TxPDO-Map Inputs Channel 1^Data In 8;
                                                            .D[9]:=TIIB[MRCO_PNL1_EP03_EP6002-0002]^COM TxPDO-Map Inputs Channel 1^Data In 9;
                                                            .D[10]:=TIIB[MRCO_PNL1_EP03_EP6002-0002]^COM TxPDO-Map Inputs Channel 1^Data In 10;
                                                            .D[11]:=TIIB[MRCO_PNL1_EP03_EP6002-0002]^COM TxPDO-Map Inputs Channel 1^Data In 11;
                                                            .D[12]:=TIIB[MRCO_PNL1_EP03_EP6002-0002]^COM TxPDO-Map Inputs Channel 1^Data In 12;
                                                            .D[13]:=TIIB[MRCO_PNL1_EP03_EP6002-0002]^COM TxPDO-Map Inputs Channel 1^Data In 13;
                                                            .D[14]:=TIIB[MRCO_PNL1_EP03_EP6002-0002]^COM TxPDO-Map Inputs Channel 1^Data In 14;
                                                            .D[15]:=TIIB[MRCO_PNL1_EP03_EP6002-0002]^COM TxPDO-Map Inputs Channel 1^Data In 15;
                                                            .D[16]:=TIIB[MRCO_PNL1_EP03_EP6002-0002]^COM TxPDO-Map Inputs Channel 1^Data In 16;
                                                            .D[17]:=TIIB[MRCO_PNL1_EP03_EP6002-0002]^COM TxPDO-Map Inputs Channel 1^Data In 17;
                                                            .D[18]:=TIIB[MRCO_PNL1_EP03_EP6002-0002]^COM TxPDO-Map Inputs Channel 1^Data In 18;
                                                            .D[19]:=TIIB[MRCO_PNL1_EP03_EP6002-0002]^COM TxPDO-Map Inputs Channel 1^Data In 19;
                                                            .D[20]:=TIIB[MRCO_PNL1_EP03_EP6002-0002]^COM TxPDO-Map Inputs Channel 1^Data In 20;
                                                            .D[21]:=TIIB[MRCO_PNL1_EP03_EP6002-0002]^COM TxPDO-Map Inputs Channel 1^Data In 21
    '}
    stComIn_MRCO_ROUGH_PTM_01        AT %I*  :       EL6inData22B;

    {attribute      'TcLinkTo'      :=      '.Ctrl:=TIIB[MRCO_PNL1_EP03_EP6002-0002]^COM RxPDO-Map Outputs Channel 1^Ctrl;
                                                            .D[0]:=TIIB[MRCO_PNL1_EP03_EP6002-0002]^COM RxPDO-Map Outputs Channel 1^Data Out 0;
                                                            .D[1]:=TIIB[MRCO_PNL1_EP03_EP6002-0002]^COM RxPDO-Map Outputs Channel 1^Data Out 1;
                                                            .D[2]:=TIIB[MRCO_PNL1_EP03_EP6002-0002]^COM RxPDO-Map Outputs Channel 1^Data Out 2;
                                                            .D[3]:=TIIB[MRCO_PNL1_EP03_EP6002-0002]^COM RxPDO-Map Outputs Channel 1^Data Out 3;
                                                            .D[4]:=TIIB[MRCO_PNL1_EP03_EP6002-0002]^COM RxPDO-Map Outputs Channel 1^Data Out 4;
                                                            .D[5]:=TIIB[MRCO_PNL1_EP03_EP6002-0002]^COM RxPDO-Map Outputs Channel 1^Data Out 5;
                                                            .D[6]:=TIIB[MRCO_PNL1_EP03_EP6002-0002]^COM RxPDO-Map Outputs Channel 1^Data Out 6;
                                                            .D[7]:=TIIB[MRCO_PNL1_EP03_EP6002-0002]^COM RxPDO-Map Outputs Channel 1^Data Out 7;
                                                            .D[8]:=TIIB[MRCO_PNL1_EP03_EP6002-0002]^COM RxPDO-Map Outputs Channel 1^Data Out 8;
                                                            .D[9]:=TIIB[MRCO_PNL1_EP03_EP6002-0002]^COM RxPDO-Map Outputs Channel 1^Data Out 9;
                                                            .D[10]:=TIIB[MRCO_PNL1_EP03_EP6002-0002]^COM RxPDO-Map Outputs Channel 1^Data Out 10;
                                                            .D[11]:=TIIB[MRCO_PNL1_EP03_EP6002-0002]^COM RxPDO-Map Outputs Channel 1^Data Out 11;
                                                            .D[12]:=TIIB[MRCO_PNL1_EP03_EP6002-0002]^COM RxPDO-Map Outputs Channel 1^Data Out 12;
                                                            .D[13]:=TIIB[MRCO_PNL1_EP03_EP6002-0002]^COM RxPDO-Map Outputs Channel 1^Data Out 13;
                                                            .D[14]:=TIIB[MRCO_PNL1_EP03_EP6002-0002]^COM RxPDO-Map Outputs Channel 1^Data Out 14;
                                                            .D[15]:=TIIB[MRCO_PNL1_EP03_EP6002-0002]^COM RxPDO-Map Outputs Channel 1^Data Out 15;
                                                            .D[16]:=TIIB[MRCO_PNL1_EP03_EP6002-0002]^COM RxPDO-Map Outputs Channel 1^Data Out 16;
                                                            .D[17]:=TIIB[MRCO_PNL1_EP03_EP6002-0002]^COM RxPDO-Map Outputs Channel 1^Data Out 17;
                                                            .D[18]:=TIIB[MRCO_PNL1_EP03_EP6002-0002]^COM RxPDO-Map Outputs Channel 1^Data Out 18;
                                                            .D[19]:=TIIB[MRCO_PNL1_EP03_EP6002-0002]^COM RxPDO-Map Outputs Channel 1^Data Out 19;
                                                            .D[20]:=TIIB[MRCO_PNL1_EP03_EP6002-0002]^COM RxPDO-Map Outputs Channel 1^Data Out 20;
                                                            .D[21]:=TIIB[MRCO_PNL1_EP03_EP6002-0002]^COM RxPDO-Map Outputs Channel 1^Data Out 21
    '}
    stComOut_MRCO_ROUGH_PTM_01        AT %Q*  :       EL6outData22B;

   {attribute	'TcLinkTo'	:=	'.Status:=TIIB[MRCO_DRL_03_E05_EL6001]^COM Inputs^Status;
                                 .D[0]:=TIIB[MRCO_DRL_03_E05_EL6001]^COM Inputs^Data In 0;
                                 .D[1]:=TIIB[MRCO_DRL_03_E05_EL6001]^COM Inputs^Data In 1;
                                 .D[2]:=TIIB[MRCO_DRL_03_E05_EL6001]^COM Inputs^Data In 2;
                                 .D[3]:=TIIB[MRCO_DRL_03_E05_EL6001]^COM Inputs^Data In 3;
                                 .D[4]:=TIIB[MRCO_DRL_03_E05_EL6001]^COM Inputs^Data In 4;
                                 .D[5]:=TIIB[MRCO_DRL_03_E05_EL6001]^COM Inputs^Data In 5;
                                 .D[6]:=TIIB[MRCO_DRL_03_E05_EL6001]^COM Inputs^Data In 6;
                                 .D[7]:=TIIB[MRCO_DRL_03_E05_EL6001]^COM Inputs^Data In 7;
                                 .D[8]:=TIIB[MRCO_DRL_03_E05_EL6001]^COM Inputs^Data In 8;
                                 .D[9]:=TIIB[MRCO_DRL_03_E05_EL6001]^COM Inputs^Data In 9;
                                 .D[10]:=TIIB[MRCO_DRL_03_E05_EL6001]^COM Inputs^Data In 10;
                                 .D[11]:=TIIB[MRCO_DRL_03_E05_EL6001]^COM Inputs^Data In 11;
                                 .D[12]:=TIIB[MRCO_DRL_03_E05_EL6001]^COM Inputs^Data In 12;
                                 .D[13]:=TIIB[MRCO_DRL_03_E05_EL6001]^COM Inputs^Data In 13;
                                 .D[14]:=TIIB[MRCO_DRL_03_E05_EL6001]^COM Inputs^Data In 14;
                                 .D[15]:=TIIB[MRCO_DRL_03_E05_EL6001]^COM Inputs^Data In 15;
                                 .D[16]:=TIIB[MRCO_DRL_03_E05_EL6001]^COM Inputs^Data In 16;
                                 .D[17]:=TIIB[MRCO_DRL_03_E05_EL6001]^COM Inputs^Data In 17;
                                 .D[18]:=TIIB[MRCO_DRL_03_E05_EL6001]^COM Inputs^Data In 18;
                                 .D[19]:=TIIB[MRCO_DRL_03_E05_EL6001]^COM Inputs^Data In 19;
                                 .D[20]:=TIIB[MRCO_DRL_03_E05_EL6001]^COM Inputs^Data In 20;
                                 .D[21]:=TIIB[MRCO_DRL_03_E05_EL6001]^COM Inputs^Data In 21
    '}
 //   stComIn_MRCO_SS_PTM_01        AT %I*  :       EL6inData22B;
     stComIn_MRCO_MSC_PTM_01        AT %I*  :       EL6inData22B;

   {attribute 'TcLinkTo'	:=	'.Ctrl:=TIIB[MRCO_DRL_03_E05_EL6001]^COM Outputs^Ctrl;
                                 .D[0]:=TIIB[MRCO_DRL_03_E05_EL6001]^COM Outputs^Data Out 0;
                                 .D[1]:=TIIB[MRCO_DRL_03_E05_EL6001]^COM Outputs^Data Out 1;
                                 .D[2]:=TIIB[MRCO_DRL_03_E05_EL6001]^COM Outputs^Data Out 2;
                                 .D[3]:=TIIB[MRCO_DRL_03_E05_EL6001]^COM Outputs^Data Out 3;
                                 .D[4]:=TIIB[MRCO_DRL_03_E05_EL6001]^COM Outputs^Data Out 4;
                                 .D[5]:=TIIB[MRCO_DRL_03_E05_EL6001]^COM Outputs^Data Out 5;
                                 .D[6]:=TIIB[MRCO_DRL_03_E05_EL6001]^COM Outputs^Data Out 6;
                                 .D[7]:=TIIB[MRCO_DRL_03_E05_EL6001]^COM Outputs^Data Out 7;
                                 .D[8]:=TIIB[MRCO_DRL_03_E05_EL6001]^COM Outputs^Data Out 8;
                                 .D[9]:=TIIB[MRCO_DRL_03_E05_EL6001]^COM Outputs^Data Out 9;
                                 .D[10]:=TIIB[MRCO_DRL_03_E05_EL6001]^COM Outputs^Data Out 10;
                                 .D[11]:=TIIB[MRCO_DRL_03_E05_EL6001]^COM Outputs^Data Out 11;
                                 .D[12]:=TIIB[MRCO_DRL_03_E05_EL6001]^COM Outputs^Data Out 12;
                                 .D[13]:=TIIB[MRCO_DRL_03_E05_EL6001]^COM Outputs^Data Out 13;
                                 .D[14]:=TIIB[MRCO_DRL_03_E05_EL6001]^COM Outputs^Data Out 14;
                                 .D[15]:=TIIB[MRCO_DRL_03_E05_EL6001]^COM Outputs^Data Out 15;
                                 .D[16]:=TIIB[MRCO_DRL_03_E05_EL6001]^COM Outputs^Data Out 16;
                                 .D[17]:=TIIB[MRCO_DRL_03_E05_EL6001]^COM Outputs^Data Out 17;
                                 .D[18]:=TIIB[MRCO_DRL_03_E05_EL6001]^COM Outputs^Data Out 18;
                                 .D[19]:=TIIB[MRCO_DRL_03_E05_EL6001]^COM Outputs^Data Out 19;
                                 .D[20]:=TIIB[MRCO_DRL_03_E05_EL6001]^COM Outputs^Data Out 20;
                                 .D[21]:=TIIB[MRCO_DRL_03_E05_EL6001]^COM Outputs^Data Out 21
    '}
 //   stComOut_MRCO_SS_PTM_01        AT %Q*  :       EL6outData22B;
    stComOut_MRCO_MSC_PTM_01        AT %Q*  :       EL6outData22B;






END_VAR

// ---- GVLs/GVL_Devices.TcGVL
//{attribute 'qualified_only'}
VAR_GLOBAL
    (*Rack Mounted Turbo Pumps*)
    {attribute 'TcLinkTo' := 	'.i_xFaultNC		:=	TIIB[MRCO_PLC_E06_EL1004]^Channel 1^Input;
                                 .i_xAtSpd  		:=	TIIB[MRCO_PLC_E06_EL1004]^Channel 2^Input;
                                 .q_RunDO			:=	TIIB[MRCO_PLC_E07_EL2794]^Channel 1^Output
    '}
    {attribute 'pytmc' := '
        pv: MRCO:MAIN:PTM:01
        io: io
    '}
    MRCO_MAIN_PTM_01 : FB_PTM_TurboDrive;

    {attribute 'TcLinkTo' := 	'.i_xFaultNC		:=	TIIB[MRCO_PLC_E06_EL1004]^Channel 3^Input;
                                 .i_xAtSpd  		:=	TIIB[MRCO_PLC_E06_EL1004]^Channel 4^Input;
                                 .q_RunDO			:=	TIIB[MRCO_PLC_E07_EL2794]^Channel 3^Output
    '}
    {attribute 'pytmc' := '
        pv: MRCO:MAIN:PTM:02
        io: io
    '}
    MRCO_MAIN_PTM_02 : FB_PTM_TurboDrive;

    {attribute 'TcLinkTo' := 	'.i_xFaultNC		:=	TIIB[MRCO_PLC_E08_EL1004]^Channel 1^Input;
                                 .i_xAtSpd  		:=	TIIB[MRCO_PLC_E08_EL1004]^Channel 2^Input;
                                 .q_RunDO			:=	TIIB[MRCO_PLC_E07_EL2794]^Channel 2^Output
    '}
    {attribute 'pytmc' := '
        pv: MRCO:MAIN:PTM:03
        io: io
    '}
    MRCO_MAIN_PTM_03 : FB_PTM_TurboDrive;

    {attribute 'TcLinkTo' := 	'.i_xFaultNC		:=	TIIB[MRCO_PLC_E08_EL1004]^Channel 3^Input;
                                 .i_xAtSpd     		:=	TIIB[MRCO_PLC_E08_EL1004]^Channel 4^Input;
                                 .q_RunDO			:=	TIIB[MRCO_PLC_E07_EL2794]^Channel 4^Output
    '}
    {attribute 'pytmc' := '
        pv: MRCO:MAIN:PTM:04
        io: io
    '}
    MRCO_MAIN_PTM_04 : FB_PTM_TurboDrive;

    (*Onboard Turbo Pumps*)

    {attribute 'TcLinkTo' := 	'.q_xReset 			:=	TIIB[MRCO_PNL1_EP02_EP2624-0002]^Channel 2^Output;
                                 .q_RunDO  			:=	TIIB[MRCO_PNL1_EP02_EP2624-0002]^Channel 1^Output;
                                 .i_xAtSpd			:=	TIIB[MRCO_PNL1_EP01_EP2338-0002]^Channel 1^Input;
                                 .i_xFaultNC		:=	TIIB[MRCO_PNL1_EP01_EP2338-0002]^Channel 2^Input
    '}
    {attribute 'pytmc' := '
        pv: MRCO:ROUGH:PTM:01
        io: io
    '}
    MRCO_ROUGH_PTM_01 : FB_PTM_Pfeiffer;

    //adding Lybold Turbovac pump MRCO-SS-PTM-01
   {attribute 'TcLinkTo' := 	'.i_xFaultNC		:=	TIIB[MRCO_DRL_03_E04_EL1004]^Channel 1^Input;
                                 .i_xAtSpd     		:=	TIIB[MRCO_DRL_03_E04_EL1004]^Channel 2^Input;
                                 .q_RunDO			:=	TIIB[MRCO_DRL_03_E06_EL2794]^Channel 1^Output
    '}
(*    {attribute 'pytmc' := '
        pv: MRCO:SS:PTM:01
        io: io
    '}

    MRCO_SS_PTM_01 : FB_PTM_TurboDrive;
    *)

    {attribute 'pytmc' := '
        pv: MRCO:MSC:PTM:01
        io: io
    '}
    MRCO_MSC_PTM_01 : FB_PTM_TurboDrive;


(*Pirani MKS 275 Gauges*)
    {attribute 'TcLinkTo' := 	'.i_iPRESS_R	:=	TIIB[MRCO_PNL1_EP05_EP3174-0002]^AI Standard Channel 1^Value
    '}
    {attribute 'pytmc' := '
        pv: MRCO:MAIN:GPI:01
        io: io
    '}
    MRCO_MAIN_GPI_01 : FB_CVM201;


(*MicroPirani MKS 925 Gauges*)
    {attribute 'TcLinkTo' := 	'.i_iPRESS_R	:=	TIIB[MRCO_PNL1_EP04_EP3174-0002]^AI Standard Channel 1^Value
    '}
    {attribute 'pytmc' := '
        pv: MRCO:ROUGH:GPI:01
        io: io
    '}
    MRCO_ROUGH_GPI_01 : FB_9XX;

    {attribute 'TcLinkTo' := 	'.i_iPRESS_R	:=	TIIB[MRCO_PNL1_EP04_EP3174-0002]^AI Standard Channel 2^Value
    '}
    {attribute 'pytmc' := '
        pv: MRCO:ROUGH:GPI:02
        io: io
    '}
    MRCO_ROUGH_GPI_02 : FB_9XX;

    {attribute 'TcLinkTo' := 	'.i_iPRESS_R	:=	TIIB[MRCO_PNL1_EP04_EP3174-0002]^AI Standard Channel 3^Value
    '}
    {attribute 'pytmc' := '
        pv: MRCO:ROUGH:GPI:03
        io: io
    '}
    MRCO_ROUGH_GPI_03 : FB_9XX;
    {attribute 'TcLinkTo' := 	'.i_iPRESS_R	:=	TIIB[MRCO_PNL1_EP04_EP3174-0002]^AI Standard Channel 4^Value
    '}
    {attribute 'pytmc' := '
        pv: MRCO:ROUGH:GPI:04
        io: io
    '}
    MRCO_ROUGH_GPI_04 : FB_9XX;

    // adding new GPI 05 for ss chamber
    {attribute 'TcLinkTo' := 	'.i_iPRESS_R	:=	TIIB[MRCO_DRL_03_E10_EL3174-0002]^AI Standard Channel 2^Value
    '}
    {attribute 'pytmc' := '
        pv: MRCO:ROUGH:GPI:05
        io: io
    '}
    MRCO_ROUGH_GPI_05 : FB_9XX;

(*Hot Cathode MKS 909 Gauges*)
    {attribute 'TcLinkTo' := 	'.i_iPRESS_R	:=	TIIB[MRCO_PNL1_EP05_EP3174-0002]^AI Standard Channel 2^Value;
                                 .q_xHV_DIS		:= 	TIIB[MRCO_PNL1_EP06_EP2624-0002]^Channel 2^Output
    '}
    {attribute 'pytmc' := '
        pv: MRCO:MAIN:GHC:01
        io: io
    '}
        MRCO_MAIN_GHC_01 : FB_MKS909;

    //adding ss chamber GHC HORNET
    {attribute 'TcLinkTo' := 	'    .i_iPRESS_R		:=	TIIB[MRCO_DRL_03_E10_EL3174-0002]^AI Standard Channel 1^Value;
                                     .i_xHV_ON			:=	TIIB[MRCO_DRL_03_E07_EL1084]^Channel 1^Input;
                                     .q_xHV_DIS			:=	TIIB[MRCO_DRL_03_E06_EL2794]^Channel 2^Output
    '}
 (*   {attribute 'pytmc' :=' pv: MRCO:SS:GHC:01'}
   MRCO_SS_GHC_01 : FB_IMG401;
   *)

    {attribute 'pytmc' :=' pv: MRCO:MSC:GHC:01'}
   MRCO_MSC_GHC_01 : FB_IMG401;


(*Variable Leak Valve*)
    {attribute 'TcLinkTo' := 	'.i_nRawPosition	:=	TIIB[VCN_1_VAT590]^DI TxPDO-Map^Position;
                                 .i_nRawPressure	:=	TIIB[VCN_1_VAT590]^DI TxPDO-Map^Pressure;
                                 .i_eControlMode	:=	TIIB[VCN_1_VAT590]^DI TxPDO-Map^Control mode;
                                 .i_eFatalError		:=	TIIB[VCN_1_VAT590]^DI TxPDO-Map^Fatal error;
                                 .i_stGenStatus 	:=	TIIB[VCN_1_VAT590]^DI TxPDO-Map^General status;
                                 .i_stGenWarnings 	:=	TIIB[VCN_1_VAT590]^DI TxPDO-Map^General warnings;
                                 .i_stExtnWarnings 	:=	TIIB[VCN_1_VAT590]^DI TxPDO-Map^Extended warnings;
                                 .o_nRawPositionSP 	:=	TIIB[VCN_1_VAT590]^DO RxPDO-Map^Position setpoint;
                                 .o_nRawPressureSP 	:=	TIIB[VCN_1_VAT590]^DO RxPDO-Map^Pressure setpoint;
                                 .o_nRawPressure 	:=	TIIB[VCN_1_VAT590]^DO RxPDO-Map^External digital pressure sensor 1;
                                 .o_eCtrlModeSP 	:=	TIIB[VCN_1_VAT590]^DO RxPDO-Map^Control mode setpoint;
                                 .o_stGenCtrlSP 	:=	TIIB[VCN_1_VAT590]^DO RxPDO-Map^General control setpoint;
                                 .i_stVat590PlcDriveRef.aNetId     := TIIB[VCN_1_VAT590]^InfoData^AdsAddr^netId;
                                 .i_stVat590PlcDriveRef.nSlaveAddr := TIIB[VCN_1_VAT590]^InfoData^AdsAddr^port;
                                 .i_bValveEthCatStatus             := TIIB[VCN_1_VAT590]^WcState^WcState
    '}
    {attribute 'pytmc' := 'pv: MRCO:VCN:01'}
    MRCO_VCN_01 : FB_VCN_VAT590;

(*Normally Closed Valve with Readback*)//ALL VALVES CURRENTLY NO
    {attribute 'TcLinkTo' := 	'.i_xOpnLS	:=	TIIB[MRCO_PNL1_EP07_EP2338-0002]^Channel 1^Input;
                                 .i_xClsLS	:=	TIIB[MRCO_PNL1_EP07_EP2338-0002]^Channel 2^Input;
                                 .q_xOPN_DO	:=	TIIB[MRCO_PNL1_EP07_EP2338-0002]^Channel 11^Output
    '}
    {attribute 'pytmc' := '
        pv: MRCO:ROUGH:VRC:01
        io: io
    '}
    MRCO_ROUGH_VRC_01 : FB_VRC;

    {attribute 'TcLinkTo' := 	'.i_xOpnLS	:=	TIIB[MRCO_PNL1_EP08_EP2338-0002]^Channel 1^Input;
                                 .i_xClsLS	:=	TIIB[MRCO_PNL1_EP08_EP2338-0002]^Channel 2^Input;
                                 .q_xOPN_DO	:=	TIIB[MRCO_PNL1_EP08_EP2338-0002]^Channel 11^Output
    '}
    {attribute 'pytmc' := '
        pv: MRCO:ROUGH:VRC:03
        io: io
    '}
    MRCO_ROUGH_VRC_03 : FB_VRC;

    (*Normally Open Valve with Readback*)

    {attribute 'TcLinkTo' := 	'.i_xOpnLS	:=	TIIB[MRCO_PNL1_EP07_EP2338-0002]^Channel 5^Input;
                                 .i_xClsLS	:=	TIIB[MRCO_PNL1_EP07_EP2338-0002]^Channel 6^Input;
                                 .q_xCLS_DO	:=	TIIB[MRCO_PNL1_EP07_EP2338-0002]^Channel 15^Output
    '}
    {attribute 'pytmc' := '
        pv: MRCO:ROUGH:VRC:02
        io: io
    '}
    MRCO_ROUGH_VRC_02 : FB_VRC_NO;



        //adding a window valve between MRCO main chamber to SS chamber
    {attribute 'TcLinkTo' := 	'.i_xOpnLS	:=	TIIB[MRCO_DRL_03_E01_EL1004]^Channel 1^Input;
                                 .i_xClsLS	:=	TIIB[MRCO_DRL_03_E01_EL1004]^Channel 2^Input;
                                 .q_xOPN_DO	:=	TIIB[MRCO_DRL_03_E02_EL2004]^Channel 1^Output
    '}
(*    {attribute 'pytmc' := '
        pv: MRCO:SS:VRC:01
        io: io
    '}
    MRCO_SS_VRC_01 : FB_VGC_2S;
    *)

    {attribute 'pytmc' := '
        pv: MRCO:MSC:VRC:01
        io: io
    '}
    MRCO_MSC_VRC_01 : FB_VGC_2S;


    //adding rough line valve in SS chamber
    {attribute 'TcLinkTo' := 	'.i_xOpnLS	:=	TIIB[MRCO_DRL_03_E01_EL1004]^Channel 3^Input;
                                 .i_xClsLS	:=	TIIB[MRCO_DRL_03_E01_EL1004]^Channel 4^Input;
                                 .q_xOPN_DO	:=	TIIB[MRCO_DRL_03_E02_EL2004]^Channel 2^Output
    '}
    {attribute 'pytmc' := '
        pv: MRCO:ROUGH:VRC:04
        io: io
    '}
    MRCO_ROUGH_VRC_04 : FB_VGC_2S;

    //adding NO valve VRC-05 in ss chamber
   {attribute 'TcLinkTo' := 	'.i_xOpnLS	:=	TIIB[MRCO_DRL_03_E03_EL1004]^Channel 1^Input;
                                 .i_xClsLS	:=	TIIB[MRCO_DRL_03_E03_EL1004]^Channel 2^Input;
                                 .q_xCLS_DO	:=	TIIB[MRCO_DRL_03_E02_EL2004]^Channel 3^Output
    '}
    {attribute 'pytmc' := '
        pv: MRCO:ROUGH:VRC:05
        io: io
    '}
    MRCO_ROUGH_VRC_05 : FB_VRC_NO;

    (*Normally Closed Valve with Readback*)

    {attribute 'TcLinkTo' := 	'.i_xOpnLS	:=	TIIB[MRCO_PNL1_EP08_EP2338-0002]^Channel 5^Input;
                                 .i_xClsLS	:=	TIIB[MRCO_PNL1_EP08_EP2338-0002]^Channel 6^Input;
                                 .q_xOPN_DO	:=	TIIB[MRCO_PNL1_EP08_EP2338-0002]^Channel 15^Output
    '}
    {attribute 'pytmc' := '
        pv: MRCO:ROUGH:VRC:06
        io: io
    '}
    MRCO_ROUGH_VRC_06 : FB_VRC;

(*Pfeiffer*)
    // They share the same serial port
    st_Pfeiffer_CTRL_MRCO_ROUGH_PTM_01   		: ARRAY[1..20] OF ST_PfeifferControl;
    st_Pfeiffer_RBK_MRCO_ROUGH_PTM_01 			: ARRAY[1..20] OF ST_PfeifferStatus;
    fb_PfeifferCom_MRCO_ROUGH_PTM_01 			: FB_PFEIFFER_COM;

(*Leybold*)
    st_TD20_RBK_MRCO_MAIN_PTM_01                : ST_TD20Status;
    fb_TD20Com_MRCO_MAIN_PTM_01                 : FB_OERLIKON_TD20_COM;

    st_TD20_RBK_MRCO_MAIN_PTM_02                : ST_TD20Status;
    fb_TD20Com_MRCO_MAIN_PTM_02                 : FB_OERLIKON_TD20_COM;

    st_TD20_RBK_MRCO_MAIN_PTM_03                : ST_TD20Status;
    fb_TD20Com_MRCO_MAIN_PTM_03                 : FB_OERLIKON_TD20_COM;

    st_TD20_RBK_MRCO_MAIN_PTM_04                : ST_TD20Status;
    fb_TD20Com_MRCO_MAIN_PTM_04                 : FB_OERLIKON_TD20_COM;

(*    st_TD400_RBK_MRCO_SS_PTM_01                : ST_TD400Status;
    fb_TD400Com_MRCO_SS_PTM_01                 : FB_OERLIKON_TD400_COM;
    st_TD400_CTRL_MRCO_SS_PTM_01               : ST_TD400Control;
    fb_TD400SerialIO_MRCO_SS_PTM_01            : FB_OERLIKON_TD400_TO_PTM;
    *)

    st_TD400_RBK_MRCO_MSC_PTM_01                : ST_TD400Status;   //need to update the library
    fb_TD400Com_MRCO_MSC_PTM_01                 : FB_OERLIKON_TD400_COM;
    st_TD400_CTRL_MRCO_MSC_PTM_01               : ST_TD400Control;
    fb_TD400SerialIO_MRCO_MSC_PTM_01            : FB_OERLIKON_TD400_TO_PTM;


END_VAR

// ---- GVLs/GVL_PLC_Interfaces.TcGVL
//{attribute 'qualified_only'}
VAR_GLOBAL

    //Outputs
    fb_ADS_WATCHDOG_VAC_MRCO_TMO:FB_ADS_WATCHDOG;
    (*ETHERCAT BRIDGE COM STATUS*)
    //0: Other side is in OP state, >0: Error
    {attribute 'TcLinkTo' := 	'TIIB[MRCO_PLC_E04_EL6695]^SYNC Inputs^TxPDO state
    '}
    xEcatBridge_TxPDO_state AT %I* : BOOL;

    //0: External device connected, 1: External device not connected
    {attribute 'TcLinkTo' := 	'TIIB[MRCO_PLC_E04_EL6695]^SYNC Inputs^External device not connected
    '}
    xEcatBridge_External_device_not_connected AT %I* : BOOL;

    //0 = Data valid, 1 = Data invalid
    {attribute 'TcLinkTo' := 	'TIIB[MRCO_PLC_E04_EL6695]^WcState^WcState
    '}
    xEcatBridge_WcState AT %I* : BOOL;

    (*I/O Inputs from TMO Beamline*)
    {attribute 'TcLinkTo' := 	'TIIB[MRCO_PLC_E04_EL6695]^IO Inputs^HUTCH_PLC_NAME
    '}
    sHUTCH_PLC_NAME AT %I* : STRING(8);

    {attribute 'TcLinkTo' := 	'TIIB[MRCO_PLC_E04_EL6695]^IO Inputs^TMO_ROUGH1_VRC_01_OPEN_LS
    '}
    xTMO_ROUGH1_VRC_01_OPEN_LS AT %I* : BOOL;

    {attribute 'TcLinkTo' := 	'TIIB[MRCO_PLC_E04_EL6695]^IO Inputs^TMO_ROUGH2_VRC_01_OPEN_LS
    '}
    xTMO_ROUGH2_VRC_01_OPEN_LS AT %I* : BOOL;


    (*I/O Outputs to TMO Beamline*)
    {attribute 'TcLinkTo' := 	'TIIB[MRCO_PLC_E04_EL6695]^IO Outputs^ENDSTATION_PLC_NAME
    '}
    sENDSTATION_PLC_NAME AT %Q* : STRING(8):= 'MRCO';

    {attribute 'TcLinkTo' := 	'TIIB[MRCO_PLC_E04_EL6695]^IO Outputs^IP1_ROUGH_VRC_01_OPEN_LS
    '}
    xIP1_ROUGH_VRC_01_OPEN_LS AT %Q* : BOOL;

    {attribute 'TcLinkTo' := 	'TIIB[MRCO_PLC_E04_EL6695]^IO Outputs^IP1_ROUGH_VRC_02_OPEN_LS
    '}
    xIP1_ROUGH_VRC_02_OPEN_LS AT %Q* : BOOL;

    {attribute 'TcLinkTo' := 	'TIIB[MRCO_PLC_E04_EL6695]^IO Outputs^IP1_ROUGH_VRC_03_OPEN_LS
    '}
    xIP1_ROUGH_VRC_03_OPEN_LS AT %Q* : BOOL;

    {attribute 'TcLinkTo' := 	'TIIB[MRCO_PLC_E04_EL6695]^IO Outputs^IP1_TURBOS_ALL_AtSpd
    '}
    {attribute 'pytmc' := '
        pv: PLC:MRCO:VAC:IP1_TURBOS_ALL_ATSPD
        io:i
    '}
    xIP1_TURBOS_ALL_AtSpd AT %Q* : BOOL;

    {attribute 'TcLinkTo' := 	'TIIB[MRCO_PLC_E04_EL6695]^IO Outputs^IP1_MAIN_xAT_VAC
    '}
    xIP1_MAIN_xAT_VAC AT %Q* : BOOL;

    {attribute 'TcLinkTo' := 	'TIIB[MRCO_PLC_E04_EL6695]^IO Outputs^IP1_MAIN_xPRESS_OK
    '}
    xIP1_MAIN_xPRESS_OK AT %Q* : BOOL;

    {attribute 'TcLinkTo' := 	'TIIB[MRCO_PLC_E04_EL6695]^IO Outputs^IP1_MAIN_rPRESS
    '}
    rIP1_MAIN_rPRESS AT %Q* : REAL;

    {attribute 'TcLinkTo' := 	'TIIB[MRCO_PLC_E04_EL6695]^IO Outputs^IP1_HV_SAFETY_ENABLE
    '}
    xIP1_HV_SAFETY_ENABLE AT %Q* : BOOL;


    (*ISEG HV Crate Safety Loop*)
    {attribute 'TcLinkTo' := 	'TIIB[MRCO_PLC_E09_EL2794]^Channel 1^Output
    '}
    {attribute 'pytmc' := '
        pv: PLC:MRCO:VAC:HV_SAFETY_ENABLE
        io:i
    '}
    xHighVoltageSafteyLoopEnable AT %Q* : BOOL := FALSE; (*When Enables the High voltage Saftey loop is closed and HV can start.*)
END_VAR

